KUKA KRL program: makrostep.src

&ACCESS RVP1
&COMMENT MAKRO_SCHRITTKETTE
&PARAM TEMPLATE = C:\KRC\Roboter\Template\makrostepvorgabe.src
&PARAM TPVW_VERSION = 8.1.8
&PARAM EDITMASK = MakroStep
DEF MAKROSTEP(Function :IN)
   ; FOLD Makro Schrittkette;%{SE} %MKUKATPVW
   ; FOLD ;%{H} %MKUKATPVW
   INT Function
   IF Function==1 THEN
     $APP_INT[5]=1
     Return
   ENDIF
   SWITCH $APP_INT[5]
   Case 0
   ; ENDFOLD
   ;ENDFOLD
   ;FOLD SCHRITT 1 -- -- ;%{P}%MKUKATPVW,%CSTEP,%VST_NR,%P 1:SCHRITT, 2:1, 3:
      ;FOLD ;%{H}
         Case 1
      ;ENDFOLD
      ;FOLD -- Roboter Schrittkette -- ;%{SE}%MKUKATPVW %CVW_COM %VCOMMENT %P 2:-- Roboter Schrittkette --, 3: VW_COMMENT
      ;ENDFOLD
      ;FOLD -- KS24 -- ;%{SE}%MKUKATPVW %CVW_COM %VCOMMENT %P 2:-- KS24 --, 3: VW_COMMENT
      ;ENDFOLD
      ;FOLD -- Version: 05 -- ;%{SE}%MKUKATPVW %CVW_COM %VCOMMENT %P 2:-- Version: 05 --, 3: VW_COMMENT
      ;ENDFOLD
      ;FOLD -- Stand: 001 -- ;%{SE}%MKUKATPVW %CVW_COM %VCOMMENT %P 2:-- Stand: 001 --, 3: VW_COMMENT
      ;ENDFOLD
      ;FOLD -- letzte Aenderung 24.10.2017 LZ -- ;%{SE}%MKUKATPVW %CVW_COM %VCOMMENT %P 2:-- letzte Aenderung 24.10.2017 LZ --, 3: VW_COMMENT
      ;ENDFOLD
      ;FOLD -- E/A's und Flags Ruecksetzen -- ;%{SE}%MKUKATPVW %CVW_COM %VCOMMENT %P 2:-- E/A's und Flags Ruecksetzen --, 3: VW_COMMENT
      ;ENDFOLD
      ;FOLD -- SK1 KF1 KS1 KE1 -- ;%{SE}%MKUKATPVW %CVW_COM %VCOMMENT %P 2:-- SK1 KF1 KS1 KE1 --, 3: VW_COMMENT
      ;ENDFOLD
      ;FOLD A786 = F830 & A786 ;%{SE}%MKUKATPVW %CVW_SPS %VBOASG %P 2:A786 = F830 & A786, 3: BOASG
         $OUT[786] = $FLAG[830] AND $OUT[786]
      ;ENDFOLD
      ;FOLD A722 = !F830 & A722 ;%{SE}%MKUKATPVW %CVW_SPS %VBOASG %P 2:A722 = !F830 & A722, 3: BOASG
         $OUT[722] = NOT $FLAG[830] AND $OUT[722]
      ;ENDFOLD
      ;FOLD A834 = AUS ;%{SE}%MKUKATPVW %CVW_SPS %VBOASG %P 2:A834 = AUS, 3: BOASG
         $OUT[834] = FALSE
      ;ENDFOLD
      ;FOLD A842 = AUS ;%{SE}%MKUKATPVW %CVW_SPS %VBOASG %P 2:A842 = AUS, 3: BOASG
         $OUT[842] = FALSE
      ;ENDFOLD
      ;FOLD -- SK2 KF2 KS2 KE2 -- ;%{SE}%MKUKATPVW %CVW_COM %VCOMMENT %P 2:-- SK2 KF2 KS2 KE2 --, 3: VW_COMMENT
      ;ENDFOLD
      ;FOLD A946 = F831 & A946 ;%{SE}%MKUKATPVW %CVW_SPS %VBOASG %P 2:A946 = F831 & A946, 3: BOASG
         $OUT[946] = $FLAG[831] AND $OUT[946]
      ;ENDFOLD
      ;FOLD A882 = !F831 & A882 ;%{SE}%MKUKATPVW %CVW_SPS %VBOASG %P 2:A882 = !F831 & A882, 3: BOASG
         $OUT[882] = NOT $FLAG[831] AND $OUT[882]
      ;ENDFOLD
      ;FOLD A994 = AUS ;%{SE}%MKUKATPVW %CVW_SPS %VBOASG %P 2:A994 = AUS, 3: BOASG
         $OUT[994] = FALSE
      ;ENDFOLD
      ;FOLD A995 = AUS ;%{SE}%MKUKATPVW %CVW_SPS %VBOASG %P 2:A995 = AUS, 3: BOASG
         $OUT[995] = FALSE
      ;ENDFOLD
      ;FOLD A1002 = AUS ;%{SE}%MKUKATPVW %CVW_SPS %VBOASG %P 2:A1002 = AUS, 3: BOASG
         $OUT[1002] = FALSE
      ;ENDFOLD
      ;FOLD -- SK3 KF3 KS3 KE3 -- ;%{SE}%MKUKATPVW %CVW_COM %VCOMMENT %P 2:-- SK3 KF3 KS3 KE3 --, 3: VW_COMMENT
      ;ENDFOLD
      ;FOLD A1106 = F832 & A1106 ;%{SE}%MKUKATPVW %CVW_SPS %VBOASG %P 2:A1106 = F832 & A1106, 3: BOASG
         $OUT[1106] = $FLAG[832] AND $OUT[1106]
      ;ENDFOLD
      ;FOLD A1042 = !F832 & A1042 ;%{SE}%MKUKATPVW %CVW_SPS %VBOASG %P 2:A1042 = !F832 & A1042, 3: BOASG
         $OUT[1042] = NOT $FLAG[832] AND $OUT[1042]
      ;ENDFOLD
      ;FOLD A1154 = AUS ;%{SE}%MKUKATPVW %CVW_SPS %VBOASG %P 2:A1154 = AUS, 3: BOASG
         $OUT[1154] = FALSE
      ;ENDFOLD
      ;FOLD A1155 = AUS ;%{SE}%MKUKATPVW %CVW_SPS %VBOASG %P 2:A1155 = AUS, 3: BOASG
         $OUT[1155] = FALSE
      ;ENDFOLD
      ;FOLD A1162 = AUS ;%{SE}%MKUKATPVW %CVW_SPS %VBOASG %P 2:A1162 = AUS, 3: BOASG
         $OUT[1162] = FALSE
      ;ENDFOLD
      ;FOLD -- Auswertung KF Umdrehungen EZ1/SP1/KE1 -- ;%{SE}%MKUKATPVW %CVW_COM %VCOMMENT %P 2:-- Auswertung KF Umdrehungen EZ1/SP1/KE1 --, 3: VW_COMMENT
      ;ENDFOLD
      ;FOLD F94 = AUS ;%{SE}%MKUKATPVW %CVW_SPS %VBOASG %P 2:F94 = AUS, 3: BOASG
         $FLAG[94] = FALSE
      ;ENDFOLD
      ;FOLD F95 = AUS ;%{SE}%MKUKATPVW %CVW_SPS %VBOASG %P 2:F95 = AUS, 3: BOASG
         $FLAG[95] = FALSE
      ;ENDFOLD
      ;FOLD F96 = AUS ;%{SE}%MKUKATPVW %CVW_SPS %VBOASG %P 2:F96 = AUS, 3: BOASG
         $FLAG[96] = FALSE
      ;ENDFOLD
      ;FOLD F97 = AUS ;%{SE}%MKUKATPVW %CVW_SPS %VBOASG %P 2:F97 = AUS, 3: BOASG
         $FLAG[97] = FALSE
      ;ENDFOLD
      ;FOLD F98 = AUS ;%{SE}%MKUKATPVW %CVW_SPS %VBOASG %P 2:F98 = AUS, 3: BOASG
         $FLAG[98] = FALSE
      ;ENDFOLD
      ;FOLD F99 = AUS ;%{SE}%MKUKATPVW %CVW_SPS %VBOASG %P 2:F99 = AUS, 3: BOASG
         $FLAG[99] = FALSE
      ;ENDFOLD
      ;FOLD F100 = AUS ;%{SE}%MKUKATPVW %CVW_SPS %VBOASG %P 2:F100 = AUS, 3: BOASG
         $FLAG[100] = FALSE
      ;ENDFOLD
      ;FOLD F101 = AUS ;%{SE}%MKUKATPVW %CVW_SPS %VBOASG %P 2:F101 = AUS, 3: BOASG
         $FLAG[101] = FALSE
      ;ENDFOLD
      ;FOLD F102 = AUS ;%{SE}%MKUKATPVW %CVW_SPS %VBOASG %P 2:F102 = AUS, 3: BOASG
         $FLAG[102] = FALSE
      ;ENDFOLD
      ;FOLD F103 = AUS ;%{SE}%MKUKATPVW %CVW_SPS %VBOASG %P 2:F103 = AUS, 3: BOASG
         $FLAG[103] = FALSE
      ;ENDFOLD
      ;FOLD F104 = AUS ;%{SE}%MKUKATPVW %CVW_SPS %VBOASG %P 2:F104 = AUS, 3: BOASG
         $FLAG[104] = FALSE
      ;ENDFOLD
      ;FOLD F105 = AUS ;%{SE}%MKUKATPVW %CVW_SPS %VBOASG %P 2:F105 = AUS, 3: BOASG
         $FLAG[105] = FALSE
      ;ENDFOLD
      ;FOLD F106 = AUS ;%{SE}%MKUKATPVW %CVW_SPS %VBOASG %P 2:F106 = AUS, 3: BOASG
         $FLAG[106] = FALSE
      ;ENDFOLD
      ;FOLD F107 = AUS ;%{SE}%MKUKATPVW %CVW_SPS %VBOASG %P 2:F107 = AUS, 3: BOASG
         $FLAG[107] = FALSE
      ;ENDFOLD
      ;FOLD F108 = AUS ;%{SE}%MKUKATPVW %CVW_SPS %VBOASG %P 2:F108 = AUS, 3: BOASG
         $FLAG[108] = FALSE
      ;ENDFOLD
      ;FOLD F109 = AUS ;%{SE}%MKUKATPVW %CVW_SPS %VBOASG %P 2:F109 = AUS, 3: BOASG
         $FLAG[109] = FALSE
      ;ENDFOLD
      ;FOLD F110 = AUS ;%{SE}%MKUKATPVW %CVW_SPS %VBOASG %P 2:F110 = AUS, 3: BOASG
         $FLAG[110] = FALSE
      ;ENDFOLD
      ;FOLD F111 = AUS ;%{SE}%MKUKATPVW %CVW_SPS %VBOASG %P 2:F111 = AUS, 3: BOASG
         $FLAG[111] = FALSE
      ;ENDFOLD
      ;FOLD F112 = AUS ;%{SE}%MKUKATPVW %CVW_SPS %VBOASG %P 2:F112 = AUS, 3: BOASG
         $FLAG[112] = FALSE
      ;ENDFOLD
      ;FOLD F113 = AUS ;%{SE}%MKUKATPVW %CVW_SPS %VBOASG %P 2:F113 = AUS, 3: BOASG
         $FLAG[113] = FALSE
      ;ENDFOLD
      ;FOLD F114 = AUS ;%{SE}%MKUKATPVW %CVW_SPS %VBOASG %P 2:F114 = AUS, 3: BOASG
         $FLAG[114] = FALSE
      ;ENDFOLD
      ;FOLD F115 = AUS ;%{SE}%MKUKATPVW %CVW_SPS %VBOASG %P 2:F115 = AUS, 3: BOASG
         $FLAG[115] = FALSE
      ;ENDFOLD
      ;FOLD F116 = AUS ;%{SE}%MKUKATPVW %CVW_SPS %VBOASG %P 2:F116 = AUS, 3: BOASG
         $FLAG[116] = FALSE
      ;ENDFOLD
      ;FOLD F117 = AUS ;%{SE}%MKUKATPVW %CVW_SPS %VBOASG %P 2:F117 = AUS, 3: BOASG
         $FLAG[117] = FALSE
      ;ENDFOLD
      ;FOLD -- Auswertung KF Umdrehungen EZ2/SP2/KE2 -- ;%{SE}%MKUKATPVW %CVW_COM %VCOMMENT %P 2:-- Auswertung KF Umdrehungen EZ2/SP2/KE2 --, 3: VW_COMMENT
      ;ENDFOLD
      ;FOLD F150 = AUS ;%{SE}%MKUKATPVW %CVW_SPS %VBOASG %P 2:F150 = AUS, 3: BOASG
         $FLAG[150] = FALSE
      ;ENDFOLD
      ;FOLD F151 = AUS ;%{SE}%MKUKATPVW %CVW_SPS %VBOASG %P 2:F151 = AUS, 3: BOASG
         $FLAG[151] = FALSE
      ;ENDFOLD
      ;FOLD F152 = AUS ;%{SE}%MKUKATPVW %CVW_SPS %VBOASG %P 2:F152 = AUS, 3: BOASG
         $FLAG[152] = FALSE
      ;ENDFOLD
      ;FOLD F153 = AUS ;%{SE}%MKUKATPVW %CVW_SPS %VBOASG %P 2:F153 = AUS, 3: BOASG
         $FLAG[153] = FALSE
      ;ENDFOLD
      ;FOLD F154 = AUS ;%{SE}%MKUKATPVW %CVW_SPS %VBOASG %P 2:F154 = AUS, 3: BOASG
         $FLAG[154] = FALSE
      ;ENDFOLD
      ;FOLD F155 = AUS ;%{SE}%MKUKATPVW %CVW_SPS %VBOASG %P 2:F155 = AUS, 3: BOASG
         $FLAG[155] = FALSE
      ;ENDFOLD
      ;FOLD -- Auswertung KF Umdrehungen EZ3/SP3/KE3 -- ;%{SE}%MKUKATPVW %CVW_COM %VCOMMENT %P 2:-- Auswertung KF Umdrehungen EZ3/SP3/KE3 --, 3: VW_COMMENT
      ;ENDFOLD
      ;FOLD F186 = AUS ;%{SE}%MKUKATPVW %CVW_SPS %VBOASG %P 2:F186 = AUS, 3: BOASG
         $FLAG[186] = FALSE
      ;ENDFOLD
      ;FOLD F187 = AUS ;%{SE}%MKUKATPVW %CVW_SPS %VBOASG %P 2:F187 = AUS, 3: BOASG
         $FLAG[187] = FALSE
      ;ENDFOLD
      ;FOLD F188 = AUS ;%{SE}%MKUKATPVW %CVW_SPS %VBOASG %P 2:F188 = AUS, 3: BOASG
         $FLAG[188] = FALSE
      ;ENDFOLD
      ;FOLD F189 = AUS ;%{SE}%MKUKATPVW %CVW_SPS %VBOASG %P 2:F189 = AUS, 3: BOASG
         $FLAG[189] = FALSE
      ;ENDFOLD
      ;FOLD F190 = AUS ;%{SE}%MKUKATPVW %CVW_SPS %VBOASG %P 2:F190 = AUS, 3: BOASG
         $FLAG[190] = FALSE
      ;ENDFOLD
      ;FOLD F191 = AUS ;%{SE}%MKUKATPVW %CVW_SPS %VBOASG %P 2:F191 = AUS, 3: BOASG
         $FLAG[191] = FALSE
      ;ENDFOLD
      ;FOLD -- Hilfsflags beim Fraesen -- ;%{SE}%MKUKATPVW %CVW_COM %VCOMMENT %P 2:-- Hilfsflags beim Fraesen --, 3: VW_COMMENT
      ;ENDFOLD
      ;FOLD F749 = AUS ;%{SE}%MKUKATPVW %CVW_SPS %VBOASG %P 2:F749 = AUS, 3: BOASG
         $FLAG[749] = FALSE
      ;ENDFOLD
      ;FOLD F287 = AUS ;%{SE}%MKUKATPVW %CVW_SPS %VBOASG %P 2:F287 = AUS, 3: BOASG
         $FLAG[287] = FALSE
      ;ENDFOLD
      ;FOLD F290 = AUS ;%{SE}%MKUKATPVW %CVW_SPS %VBOASG %P 2:F290 = AUS, 3: BOASG
         $FLAG[290] = FALSE
      ;ENDFOLD
      ;FOLD F291 = AUS ;%{SE}%MKUKATPVW %CVW_SPS %VBOASG %P 2:F291 = AUS, 3: BOASG
         $FLAG[291] = FALSE
      ;ENDFOLD
      ;FOLD -- Hilfsflags SZ2 an SK1 -- ;%{SE}%MKUKATPVW %CVW_COM %VCOMMENT %P 2:-- Hilfsflags SZ2 an SK1 --, 3: VW_COMMENT
      ;ENDFOLD
      ;FOLD F307 = AUS ;%{SE}%MKUKATPVW %CVW_SPS %VBOASG %P 2:F307 = AUS, 3: BOASG
         $FLAG[307] = FALSE
      ;ENDFOLD
      ;FOLD F308 = AUS ;%{SE}%MKUKATPVW %CVW_SPS %VBOASG %P 2:F308 = AUS, 3: BOASG
         $FLAG[308] = FALSE
      ;ENDFOLD
      ;FOLD -- Hilfsflags Funktionstest KF Motor -- ;%{SE}%MKUKATPVW %CVW_COM %VCOMMENT %P 2:-- Hilfsflags Funktionstest KF Motor --, 3: VW_COMMENT
      ;ENDFOLD
      ;FOLD F312 = AUS ;%{SE}%MKUKATPVW %CVW_SPS %VBOASG %P 2:F312 = AUS, 3: BOASG
         $FLAG[312] = FALSE
      ;ENDFOLD
      ;FOLD F313 = AUS ;%{SE}%MKUKATPVW %CVW_SPS %VBOASG %P 2:F313 = AUS, 3: BOASG
         $FLAG[313] = FALSE
      ;ENDFOLD
      ;FOLD -- RSK Fehlerausgaben -- ;%{SE}%MKUKATPVW %CVW_COM %VCOMMENT %P 2:-- RSK Fehlerausgaben --, 3: VW_COMMENT
      ;ENDFOLD
      ;FOLD F322 = AUS ;%{SE}%MKUKATPVW %CVW_SPS %VBOASG %P 2:F322 = AUS, 3: BOASG
         $FLAG[322] = FALSE
      ;ENDFOLD
      ;FOLD F323 = AUS ;%{SE}%MKUKATPVW %CVW_SPS %VBOASG %P 2:F323 = AUS, 3: BOASG
         $FLAG[323] = FALSE
      ;ENDFOLD
      ;FOLD F324 = AUS ;%{SE}%MKUKATPVW %CVW_SPS %VBOASG %P 2:F324 = AUS, 3: BOASG
         $FLAG[324] = FALSE
      ;ENDFOLD
      ;FOLD F325 = AUS ;%{SE}%MKUKATPVW %CVW_SPS %VBOASG %P 2:F325 = AUS, 3: BOASG
         $FLAG[325] = FALSE
      ;ENDFOLD
      ;FOLD F326 = AUS ;%{SE}%MKUKATPVW %CVW_SPS %VBOASG %P 2:F326 = AUS, 3: BOASG
         $FLAG[326] = FALSE
      ;ENDFOLD
      ;FOLD F327 = AUS ;%{SE}%MKUKATPVW %CVW_SPS %VBOASG %P 2:F327 = AUS, 3: BOASG
         $FLAG[327] = FALSE
      ;ENDFOLD
      ;FOLD F328 = AUS ;%{SE}%MKUKATPVW %CVW_SPS %VBOASG %P 2:F328 = AUS, 3: BOASG
         $FLAG[328] = FALSE
      ;ENDFOLD
      ;FOLD F329 = AUS ;%{SE}%MKUKATPVW %CVW_SPS %VBOASG %P 2:F329 = AUS, 3: BOASG
         $FLAG[329] = FALSE
      ;ENDFOLD
      ;FOLD -- Hilfsflag SK Programmwechsel -- ;%{SE}%MKUKATPVW %CVW_COM %VCOMMENT %P 2:-- Hilfsflag SK Programmwechsel --, 3: VW_COMMENT
      ;ENDFOLD
      ;FOLD F334 = AUS ;%{SE}%MKUKATPVW %CVW_SPS %VBOASG %P 2:F334 = AUS, 3: BOASG
         $FLAG[334] = FALSE
      ;ENDFOLD
      ;FOLD -- Flag KL1 Spueleimer -- ;%{SE}%MKUKATPVW %CVW_COM %VCOMMENT %P 2:-- Flag KL1 Spueleimer --, 3: VW_COMMENT
      ;ENDFOLD
      ;FOLD F352 = AUS ;%{SE}%MKUKATPVW %CVW_SPS %VBOASG %P 2:F352 = AUS, 3: BOASG
         $FLAG[352] = FALSE
      ;ENDFOLD
      ;FOLD F353 = AUS ;%{SE}%MKUKATPVW %CVW_SPS %VBOASG %P 2:F353 = AUS, 3: BOASG
         $FLAG[353] = FALSE
      ;ENDFOLD
      ;FOLD -- Flag KL2 Spueleimer -- ;%{SE}%MKUKATPVW %CVW_COM %VCOMMENT %P 2:-- Flag KL2 Spueleimer --, 3: VW_COMMENT
      ;ENDFOLD
      ;FOLD F373 = AUS ;%{SE}%MKUKATPVW %CVW_SPS %VBOASG %P 2:F373 = AUS, 3: BOASG
         $FLAG[373] = FALSE
      ;ENDFOLD
      ;FOLD F374 = AUS ;%{SE}%MKUKATPVW %CVW_SPS %VBOASG %P 2:F374 = AUS, 3: BOASG
         $FLAG[374] = FALSE
      ;ENDFOLD
      ;FOLD -- Flag KL3 Spueleimer -- ;%{SE}%MKUKATPVW %CVW_COM %VCOMMENT %P 2:-- Flag KL3 Spueleimer --, 3: VW_COMMENT
      ;ENDFOLD
      ;FOLD F394 = AUS ;%{SE}%MKUKATPVW %CVW_SPS %VBOASG %P 2:F394 = AUS, 3: BOASG
         $FLAG[394] = FALSE
      ;ENDFOLD
      ;FOLD F395 = AUS ;%{SE}%MKUKATPVW %CVW_SPS %VBOASG %P 2:F395 = AUS, 3: BOASG
         $FLAG[395] = FALSE
      ;ENDFOLD
      ;FOLD -- Flag MS Reinigung gestartet -- ;%{SE}%MKUKATPVW %CVW_COM %VCOMMENT %P 2:-- Flag MS Reinigung gestartet --, 3: VW_COMMENT
      ;ENDFOLD
      ;FOLD F604 = AUS ;%{SE}%MKUKATPVW %CVW_SPS %VBOASG %P 2:F604 = AUS, 3: BOASG
         $FLAG[604] = FALSE
      ;ENDFOLD
      ;FOLD F608 = AUS ;%{SE}%MKUKATPVW %CVW_SPS %VBOASG %P 2:F608 = AUS, 3: BOASG
         $FLAG[608] = FALSE
      ;ENDFOLD
      ;FOLD -- Timer Stoppen -- ;%{SE}%MKUKATPVW %CVW_COM %VCOMMENT %P 2:-- Timer Stoppen --, 3: VW_COMMENT
      ;ENDFOLD
      ;FOLD t7 ( EIN ) = STOP ;%{SE}%MKUKATPVW %CVW_SPS %VTSTOP %P 2:t7 ( EIN ) = STOP, 3: TSTOP
         VW(#SET_TIME,TRUE,7,1,0)
      ;ENDFOLD
      ;FOLD t8 ( EIN ) = STOP ;%{SE}%MKUKATPVW %CVW_SPS %VTSTOP %P 2:t8 ( EIN ) = STOP, 3: TSTOP
         VW(#SET_TIME,TRUE,8,1,0)
      ;ENDFOLD
      ;FOLD t9 ( EIN ) = STOP ;%{SE}%MKUKATPVW %CVW_SPS %VTSTOP %P 2:t9 ( EIN ) = STOP, 3: TSTOP
         VW(#SET_TIME,TRUE,9,1,0)
      ;ENDFOLD
      ;FOLD Schritt 2 = EIN  ;%{SE}%MKUKATPVW %CVW_SPS %VST_CON %P 2:Schritt 2 = EIN , 3: ST_CON
         IF TRUE THEN
            PREVSTEP = $APP_INT[5]
            $APP_INT[5] = 2
         ENDIF
      ;ENDFOLD
   ;ENDFOLD
   ;FOLD SCHRITT 2 -- RSK Grundstellung # Anwahlen-- ;%{P}%MKUKATPVW,%CSTEP,%VST_NR,%P 1:SCHRITT, 2:2, 3: RSK Grundstellung # Anwahlen
      ;FOLD ;%{H}
         Case 2
      ;ENDFOLD
      ;FOLD -- RSK in Grundstellung -- ;%{SE}%MKUKATPVW %CVW_COM %VCOMMENT %P 2:-- RSK in Grundstellung --, 3: VW_COMMENT
      ;ENDFOLD
      ;FOLD F321 = EIN ;%{SE}%MKUKATPVW %CVW_SPS %VBOASG %P 2:F321 = EIN, 3: BOASG
         $FLAG[321] = TRUE
      ;ENDFOLD
      ;FOLD -- Fraesen ROB EZ1/SP1/KE1 SZ1 (Basic/Docking) -- ;%{SE}%MKUKATPVW %CVW_COM %VCOMMENT %P 2:-- Fraesen ROB EZ1/SP1/KE1 SZ1 (Basic/Docking) --, 3: VW_COMMENT
      ;ENDFOLD
      ;FOLD Schritt 3 = F64 & !F65 & !F66 & !F67 & F90 & !F91 & !F565 & A4039  ;%{SE}%MKUKATPVW %CVW_SPS %VST_CON %P 2:Schritt 3 = F64 & !F65 & !F66 & !F67 & F90 & !F91 & !F565 & A4039 , 3: ST_CON
         IF $FLAG[64] AND NOT $FLAG[65] AND NOT $FLAG[66] AND NOT $FLAG[67] AND $FLAG[90] AND NOT $FLAG[91] AND NOT $FLAG[565] AND $OUT[4039] THEN
            PREVSTEP = $APP_INT[5]
            $APP_INT[5] = 3
         ENDIF
      ;ENDFOLD
      ;FOLD -- Fraesen ROB EZ1/SP1/KE1 SZ2 (Docking) -- ;%{SE}%MKUKATPVW %CVW_COM %VCOMMENT %P 2:-- Fraesen ROB EZ1/SP1/KE1 SZ2 (Docking) --, 3: VW_COMMENT
      ;ENDFOLD
      ;FOLD Schritt 15 = !F64 & F65 & !F66 & !F67 & F90 & !F91 & !F565 & A4039  ;%{SE}%MKUKATPVW %CVW_SPS %VST_CON %P 2:Schritt 15 = !F64 & F65 & !F66 & !F67 & F90 & !F91 & !F565 & A4039 , 3: ST_CON
         IF NOT $FLAG[64] AND $FLAG[65] AND NOT $FLAG[66] AND NOT $FLAG[67] AND $FLAG[90] AND NOT $FLAG[91] AND NOT $FLAG[565] AND $OUT[4039] THEN
            PREVSTEP = $APP_INT[5]
            $APP_INT[5] = 15
         ENDIF
      ;ENDFOLD
      ;FOLD -- Fraesen ROB EZ1/SP1/KE1 SZ3 (Docking) -- ;%{SE}%MKUKATPVW %CVW_COM %VCOMMENT %P 2:-- Fraesen ROB EZ1/SP1/KE1 SZ3 (Docking) --, 3: VW_COMMENT
      ;ENDFOLD
      ;FOLD Schritt 27 = !F64 & !F65 & F66 & !F67 & F90 & !F91 & !F565 & A4039  ;%{SE}%MKUKATPVW %CVW_SPS %VST_CON %P 2:Schritt 27 = !F64 & !F65 & F66 & !F67 & F90 & !F91 & !F565 & A4039 , 3: ST_CON
         IF NOT $FLAG[64] AND NOT $FLAG[65] AND $FLAG[66] AND NOT $FLAG[67] AND $FLAG[90] AND NOT $FLAG[91] AND NOT $FLAG[565] AND $OUT[4039] THEN
            PREVSTEP = $APP_INT[5]
            $APP_INT[5] = 27
         ENDIF
      ;ENDFOLD
      ;FOLD -- Fraesen ROB EZ1/SP1/KE1 SZ4 (Docking) -- ;%{SE}%MKUKATPVW %CVW_COM %VCOMMENT %P 2:-- Fraesen ROB EZ1/SP1/KE1 SZ4 (Docking) --, 3: VW_COMMENT
      ;ENDFOLD
      ;FOLD Schritt 39 = !F64 & !F65 & !F66 & F67 & F90 & !F91 & !F565 & A4039  ;%{SE}%MKUKATPVW %CVW_SPS %VST_CON %P 2:Schritt 39 = !F64 & !F65 & !F66 & F67 & F90 & !F91 & !F565 & A4039 , 3: ST_CON
         IF NOT $FLAG[64] AND NOT $FLAG[65] AND NOT $FLAG[66] AND $FLAG[67] AND $FLAG[90] AND NOT $FLAG[91] AND NOT $FLAG[565] AND $OUT[4039] THEN
            PREVSTEP = $APP_INT[5]
            $APP_INT[5] = 39
         ENDIF
      ;ENDFOLD
      ;FOLD -- Fraesen STAT EZ1/SP1/KE1 -- ;%{SE}%MKUKATPVW %CVW_COM %VCOMMENT %P 2:-- Fraesen STAT EZ1/SP1/KE1 --, 3: VW_COMMENT
      ;ENDFOLD
      ;FOLD Schritt 51 = F92 & !F93 & A4039 & E13  ;%{SE}%MKUKATPVW %CVW_SPS %VST_CON %P 2:Schritt 51 = F92 & !F93 & A4039 & E13 , 3: ST_CON
         IF $FLAG[92] AND NOT $FLAG[93] AND $OUT[4039] AND $IN[13] THEN
            PREVSTEP = $APP_INT[5]
            $APP_INT[5] = 51
         ENDIF
      ;ENDFOLD
      ;FOLD -- Fraesen STAT EZ2/SP2/KE2 -- ;%{SE}%MKUKATPVW %CVW_COM %VCOMMENT %P 2:-- Fraesen STAT EZ2/SP2/KE2 --, 3: VW_COMMENT
      ;ENDFOLD
      ;FOLD Schritt 74 = F148 & !F149 & A4039 & E13  ;%{SE}%MKUKATPVW %CVW_SPS %VST_CON %P 2:Schritt 74 = F148 & !F149 & A4039 & E13 , 3: ST_CON
         IF $FLAG[148] AND NOT $FLAG[149] AND $OUT[4039] AND $IN[13] THEN
            PREVSTEP = $APP_INT[5]
            $APP_INT[5] = 74
         ENDIF
      ;ENDFOLD
      ;FOLD -- Fraesen STAT EZ3/SP3/KE3 -- ;%{SE}%MKUKATPVW %CVW_COM %VCOMMENT %P 2:-- Fraesen STAT EZ3/SP3/KE3 --, 3: VW_COMMENT
      ;ENDFOLD
      ;FOLD Schritt 97 = F184 & !F185 & A4039 & E13  ;%{SE}%MKUKATPVW %CVW_SPS %VST_CON %P 2:Schritt 97 = F184 & !F185 & A4039 & E13 , 3: ST_CON
         IF $FLAG[184] AND NOT $FLAG[185] AND $OUT[4039] AND $IN[13] THEN
            PREVSTEP = $APP_INT[5]
            $APP_INT[5] = 97
         ENDIF
      ;ENDFOLD
      ;FOLD -- Fraesen ROB STP1 SZ1 (Stosspunkten) -- ;%{SE}%MKUKATPVW %CVW_COM %VCOMMENT %P 2:-- Fraesen ROB STP1 SZ1 (Stosspunkten) --, 3: VW_COMMENT
      ;ENDFOLD
      ;FOLD Schritt 120 = F64 & !F65 & !F66 & !F67 & F90 & !F91 & !F805 & F565 & A4039 & E13  ;%{SE}%MKUKATPVW %CVW_SPS %VST_CON %P 2:Schritt 120 = F64 & !F65 & !F66 & !F67 & F90 & !F91 & !F805 & F565 & A4039 & E13 , 3: ST_CON
         IF $FLAG[64] AND NOT $FLAG[65] AND NOT $FLAG[66] AND NOT $FLAG[67] AND $FLAG[90] AND NOT $FLAG[91] AND NOT $FLAG[805] AND $FLAG[565] AND $OUT[4039] AND $IN[13] THEN
            PREVSTEP = $APP_INT[5]
            $APP_INT[5] = 120
         ENDIF
      ;ENDFOLD
      ;FOLD -- MS1 Reinigung (an KS3 Schwenkeinheit) -- ;%{SE}%MKUKATPVW %CVW_COM %VCOMMENT %P 2:-- MS1 Reinigung (an KS3 Schwenkeinheit) --, 3: VW_COMMENT
      ;ENDFOLD
      ;FOLD Schritt 128 = F603 & !F605 & F528 & !F529 & A4039 & E13  ;%{SE}%MKUKATPVW %CVW_SPS %VST_CON %P 2:Schritt 128 = F603 & !F605 & F528 & !F529 & A4039 & E13 , 3: ST_CON
         IF $FLAG[603] AND NOT $FLAG[605] AND $FLAG[528] AND NOT $FLAG[529] AND $OUT[4039] AND $IN[13] THEN
            PREVSTEP = $APP_INT[5]
            $APP_INT[5] = 128
         ENDIF
      ;ENDFOLD
      ;FOLD -- MS2 Reinigung (an KS2 Schwenkeinheit) -- ;%{SE}%MKUKATPVW %CVW_COM %VCOMMENT %P 2:-- MS2 Reinigung (an KS2 Schwenkeinheit) --, 3: VW_COMMENT
      ;ENDFOLD
      ;FOLD Schritt 141 = F607 & !F609 & F528 & !F529 & A4039 & E13  ;%{SE}%MKUKATPVW %CVW_SPS %VST_CON %P 2:Schritt 141 = F607 & !F609 & F528 & !F529 & A4039 & E13 , 3: ST_CON
         IF $FLAG[607] AND NOT $FLAG[609] AND $FLAG[528] AND NOT $FLAG[529] AND $OUT[4039] AND $IN[13] THEN
            PREVSTEP = $APP_INT[5]
            $APP_INT[5] = 141
         ENDIF
      ;ENDFOLD
      ;FOLD -- MS1 Reinigung (an Pneum. Schwenkeinheit MS1) -- ;%{SE}%MKUKATPVW %CVW_COM %VCOMMENT %P 2:-- MS1 Reinigung (an Pneum. Schwenkeinheit MS1) --, 3: VW_COMMENT
      ;ENDFOLD
      ;FOLD Schritt 154 = F603 & !F605 & !F528 & F529 & A4039 & E13  ;%{SE}%MKUKATPVW %CVW_SPS %VST_CON %P 2:Schritt 154 = F603 & !F605 & !F528 & F529 & A4039 & E13 , 3: ST_CON
         IF $FLAG[603] AND NOT $FLAG[605] AND NOT $FLAG[528] AND $FLAG[529] AND $OUT[4039] AND $IN[13] THEN
            PREVSTEP = $APP_INT[5]
            $APP_INT[5] = 154
         ENDIF
      ;ENDFOLD
      ;FOLD -- MS2 Reinigung (an Pneum. Schwenkeinheit MS2) -- ;%{SE}%MKUKATPVW %CVW_COM %VCOMMENT %P 2:-- MS2 Reinigung (an Pneum. Schwenkeinheit MS2) --, 3: VW_COMMENT
      ;ENDFOLD
      ;FOLD Schritt 169 = F607 & !F609 & !F528 & F529 & A4039 & E13  ;%{SE}%MKUKATPVW %CVW_SPS %VST_CON %P 2:Schritt 169 = F607 & !F609 & !F528 & F529 & A4039 & E13 , 3: ST_CON
         IF $FLAG[607] AND NOT $FLAG[609] AND NOT $FLAG[528] AND $FLAG[529] AND $OUT[4039] AND $IN[13] THEN
            PREVSTEP = $APP_INT[5]
            $APP_INT[5] = 169
         ENDIF
      ;ENDFOLD
      ;FOLD -- KL1 Spueleimer (an Pneum. Schwenkeinheit KL1) -- ;%{SE}%MKUKATPVW %CVW_COM %VCOMMENT %P 2:-- KL1 Spueleimer (an Pneum. Schwenkeinheit KL1) --, 3: VW_COMMENT
      ;ENDFOLD
      ;FOLD -- in Arbeitsstellung schwenken -- ;%{SE}%MKUKATPVW %CVW_COM %VCOMMENT %P 2:-- in Arbeitsstellung schwenken --, 3: VW_COMMENT
      ;ENDFOLD
      ;FOLD Schritt 184 = !F352 & F353 & !F355 & (F523 & !F524 + !F523 & F524) & A4039 & E13  ;%{SE}%MKUKATPVW %CVW_SPS %VST_CON %P 2:Schritt 184 = !F352 & F353 & !F355 & (F523 & !F524 + !F523 & F524) & A4039 & E13 , 3: ST_CON
         IF NOT $FLAG[352] AND $FLAG[353] AND NOT $FLAG[355] AND ($FLAG[523] AND NOT $FLAG[524] OR NOT $FLAG[523] AND $FLAG[524]) AND $OUT[4039] AND $IN[13] THEN
            PREVSTEP = $APP_INT[5]
            $APP_INT[5] = 184
         ENDIF
      ;ENDFOLD
      ;FOLD -- KL1 Spueleimer (an Pneum. Schwenkeinheit KL1) -- ;%{SE}%MKUKATPVW %CVW_COM %VCOMMENT %P 2:-- KL1 Spueleimer (an Pneum. Schwenkeinheit KL1) --, 3: VW_COMMENT
      ;ENDFOLD
      ;FOLD -- in Ruhestellung schwenken -- ;%{SE}%MKUKATPVW %CVW_COM %VCOMMENT %P 2:-- in Ruhestellung schwenken --, 3: VW_COMMENT
      ;ENDFOLD
      ;FOLD Schritt 189 = F352 & !F353 & !F355 & (F523 & !F524 + !F523 & F524) & A4039 & E13  ;%{SE}%MKUKATPVW %CVW_SPS %VST_CON %P 2:Schritt 189 = F352 & !F353 & !F355 & (F523 & !F524 + !F523 & F524) & A4039 & E13 , 3: ST_CON
         IF $FLAG[352] AND NOT $FLAG[353] AND NOT $FLAG[355] AND ($FLAG[523] AND NOT $FLAG[524] OR NOT $FLAG[523] AND $FLAG[524]) AND $OUT[4039] AND $IN[13] THEN
            PREVSTEP = $APP_INT[5]
            $APP_INT[5] = 189
         ENDIF
      ;ENDFOLD
      ;FOLD -- KL2 Spueleimer (an Pneum. Schwenkeinheit KL2) -- ;%{SE}%MKUKATPVW %CVW_COM %VCOMMENT %P 2:-- KL2 Spueleimer (an Pneum. Schwenkeinheit KL2) --, 3: VW_COMMENT
      ;ENDFOLD
      ;FOLD -- in Arbeitsstellung schwenken -- ;%{SE}%MKUKATPVW %CVW_COM %VCOMMENT %P 2:-- in Arbeitsstellung schwenken --, 3: VW_COMMENT
      ;ENDFOLD
      ;FOLD Schritt 195 = !F373 & F374 & !F376 & (F523 & !F524 + !F523 & F524) & A4039 & E13  ;%{SE}%MKUKATPVW %CVW_SPS %VST_CON %P 2:Schritt 195 = !F373 & F374 & !F376 & (F523 & !F524 + !F523 & F524) & A4039 & E13 , 3: ST_CON
         IF NOT $FLAG[373] AND $FLAG[374] AND NOT $FLAG[376] AND ($FLAG[523] AND NOT $FLAG[524] OR NOT $FLAG[523] AND $FLAG[524]) AND $OUT[4039] AND $IN[13] THEN
            PREVSTEP = $APP_INT[5]
            $APP_INT[5] = 195
         ENDIF
      ;ENDFOLD
      ;FOLD -- KL2 Spueleimer (an Pneum. Schwenkeinheit KL2) -- ;%{SE}%MKUKATPVW %CVW_COM %VCOMMENT %P 2:-- KL2 Spueleimer (an Pneum. Schwenkeinheit KL2) --, 3: VW_COMMENT
      ;ENDFOLD
      ;FOLD -- in Ruhestellung schwenken -- ;%{SE}%MKUKATPVW %CVW_COM %VCOMMENT %P 2:-- in Ruhestellung schwenken --, 3: VW_COMMENT
      ;ENDFOLD
      ;FOLD Schritt 200 = F373 & !F374 & !F376 & (F523 & !F524 + !F523 & F524) & A4039 & E13  ;%{SE}%MKUKATPVW %CVW_SPS %VST_CON %P 2:Schritt 200 = F373 & !F374 & !F376 & (F523 & !F524 + !F523 & F524) & A4039 & E13 , 3: ST_CON
         IF $FLAG[373] AND NOT $FLAG[374] AND NOT $FLAG[376] AND ($FLAG[523] AND NOT $FLAG[524] OR NOT $FLAG[523] AND $FLAG[524]) AND $OUT[4039] AND $IN[13] THEN
            PREVSTEP = $APP_INT[5]
            $APP_INT[5] = 200
         ENDIF
      ;ENDFOLD
      ;FOLD -- KL3 Spueleimer (an Pneum. Schwenkeinheit KL3) -- ;%{SE}%MKUKATPVW %CVW_COM %VCOMMENT %P 2:-- KL3 Spueleimer (an Pneum. Schwenkeinheit KL3) --, 3: VW_COMMENT
      ;ENDFOLD
      ;FOLD -- in Arbeitsstellung schwenken -- ;%{SE}%MKUKATPVW %CVW_COM %VCOMMENT %P 2:-- in Arbeitsstellung schwenken --, 3: VW_COMMENT
      ;ENDFOLD
      ;FOLD Schritt 206 = !F394 & F395 & !F397 & (F523 & !F524 + !F523 & F524) & A4039 & E13  ;%{SE}%MKUKATPVW %CVW_SPS %VST_CON %P 2:Schritt 206 = !F394 & F395 & !F397 & (F523 & !F524 + !F523 & F524) & A4039 & E13 , 3: ST_CON
         IF NOT $FLAG[394] AND $FLAG[395] AND NOT $FLAG[397] AND ($FLAG[523] AND NOT $FLAG[524] OR NOT $FLAG[523] AND $FLAG[524]) AND $OUT[4039] AND $IN[13] THEN
            PREVSTEP = $APP_INT[5]
            $APP_INT[5] = 206
         ENDIF
      ;ENDFOLD
      ;FOLD -- KL3 Spueleimer (an Pneum. Schwenkeinheit KL3) -- ;%{SE}%MKUKATPVW %CVW_COM %VCOMMENT %P 2:-- KL3 Spueleimer (an Pneum. Schwenkeinheit KL3) --, 3: VW_COMMENT
      ;ENDFOLD
      ;FOLD -- in Ruhestellung schwenken -- ;%{SE}%MKUKATPVW %CVW_COM %VCOMMENT %P 2:-- in Ruhestellung schwenken --, 3: VW_COMMENT
      ;ENDFOLD
      ;FOLD Schritt 211 = F394 & !F395 & !F397 & (F523 & !F524 + !F523 & F524) & A4039 & E13  ;%{SE}%MKUKATPVW %CVW_SPS %VST_CON %P 2:Schritt 211 = F394 & !F395 & !F397 & (F523 & !F524 + !F523 & F524) & A4039 & E13 , 3: ST_CON
         IF $FLAG[394] AND NOT $FLAG[395] AND NOT $FLAG[397] AND ($FLAG[523] AND NOT $FLAG[524] OR NOT $FLAG[523] AND $FLAG[524]) AND $OUT[4039] AND $IN[13] THEN
            PREVSTEP = $APP_INT[5]
            $APP_INT[5] = 211
         ENDIF
      ;ENDFOLD
      ;FOLD -- Fraesen MB1 (an KSB1 Schwenkeinheit) -- ;%{SE}%MKUKATPVW %CVW_COM %VCOMMENT %P 2:-- Fraesen MB1 (an KSB1 Schwenkeinheit) --, 3: VW_COMMENT
      ;ENDFOLD
      ;FOLD Schritt 250 = F209 & !F210 & A4039 & E13  ;%{SE}%MKUKATPVW %CVW_SPS %VST_CON %P 2:Schritt 250 = F209 & !F210 & A4039 & E13 , 3: ST_CON
         IF $FLAG[209] AND NOT $FLAG[210] AND $OUT[4039] AND $IN[13] THEN
            PREVSTEP = $APP_INT[5]
            $APP_INT[5] = 250
         ENDIF
      ;ENDFOLD
      ;FOLD -- Fraesen ROB STP1 SZ1 (Stosspunkten & KW Braeuer) -- ;%{SE}%MKUKATPVW %CVW_COM %VCOMMENT %P 2:-- Fraesen ROB STP1 SZ1 (Stosspunkten & KW Braeuer) --, 3: VW_COMMENT
      ;ENDFOLD
      ;FOLD Schritt 272 = F64 & !F65 & !F66 & !F67 & F90 & !F91 & F805 & F565 & A4039  ;%{SE}%MKUKATPVW %CVW_SPS %VST_CON %P 2:Schritt 272 = F64 & !F65 & !F66 & !F67 & F90 & !F91 & F805 & F565 & A4039 , 3: ST_CON
         IF $FLAG[64] AND NOT $FLAG[65] AND NOT $FLAG[66] AND NOT $FLAG[67] AND $FLAG[90] AND NOT $FLAG[91] AND $FLAG[805] AND $FLAG[565] AND $OUT[4039] THEN
            PREVSTEP = $APP_INT[5]
            $APP_INT[5] = 272
         ENDIF
      ;ENDFOLD
   ;ENDFOLD
   ;FOLD SCHRITT 3 -- ROB EZ1/SP1/KE1 SZ1 # Start -- ;%{P}%MKUKATPVW,%CSTEP,%VST_NR,%P 1:SCHRITT, 2:3, 3: ROB EZ1/SP1/KE1 SZ1 # Start
      ;FOLD ;%{H}
         Case 3
      ;ENDFOLD
      ;FOLD -- RSK gestartet -- ;%{SE}%MKUKATPVW %CVW_COM %VCOMMENT %P 2:-- RSK gestartet --, 3: VW_COMMENT
      ;ENDFOLD
      ;FOLD F321 = AUS ;%{SE}%MKUKATPVW %CVW_SPS %VBOASG %P 2:F321 = AUS, 3: BOASG
         $FLAG[321] = FALSE
      ;ENDFOLD
      ;FOLD F322 = AUS ;%{SE}%MKUKATPVW %CVW_SPS %VBOASG %P 2:F322 = AUS, 3: BOASG
         $FLAG[322] = FALSE
      ;ENDFOLD
      ;FOLD F323 = AUS ;%{SE}%MKUKATPVW %CVW_SPS %VBOASG %P 2:F323 = AUS, 3: BOASG
         $FLAG[323] = FALSE
      ;ENDFOLD
      ;FOLD F324 = AUS ;%{SE}%MKUKATPVW %CVW_SPS %VBOASG %P 2:F324 = AUS, 3: BOASG
         $FLAG[324] = FALSE
      ;ENDFOLD
      ;FOLD F325 = AUS ;%{SE}%MKUKATPVW %CVW_SPS %VBOASG %P 2:F325 = AUS, 3: BOASG
         $FLAG[325] = FALSE
      ;ENDFOLD
      ;FOLD F327 = AUS ;%{SE}%MKUKATPVW %CVW_SPS %VBOASG %P 2:F327 = AUS, 3: BOASG
         $FLAG[327] = FALSE
      ;ENDFOLD
      ;FOLD F329 = AUS ;%{SE}%MKUKATPVW %CVW_SPS %VBOASG %P 2:F329 = AUS, 3: BOASG
         $FLAG[329] = FALSE
      ;ENDFOLD
      ;FOLD -- EZ1/SP1/KE1 SZ1 Zaehler -- ;%{SE}%MKUKATPVW %CVW_COM %VCOMMENT %P 2:-- EZ1/SP1/KE1 SZ1 Zaehler --, 3: VW_COMMENT
      ;ENDFOLD
      ;FOLD F94 = AUS ;%{SE}%MKUKATPVW %CVW_SPS %VBOASG %P 2:F94 = AUS, 3: BOASG
         $FLAG[94] = FALSE
      ;ENDFOLD
      ;FOLD F95 = AUS ;%{SE}%MKUKATPVW %CVW_SPS %VBOASG %P 2:F95 = AUS, 3: BOASG
         $FLAG[95] = FALSE
      ;ENDFOLD
      ;FOLD F96 = AUS ;%{SE}%MKUKATPVW %CVW_SPS %VBOASG %P 2:F96 = AUS, 3: BOASG
         $FLAG[96] = FALSE
      ;ENDFOLD
      ;FOLD F97 = AUS ;%{SE}%MKUKATPVW %CVW_SPS %VBOASG %P 2:F97 = AUS, 3: BOASG
         $FLAG[97] = FALSE
      ;ENDFOLD
      ;FOLD F98 = AUS ;%{SE}%MKUKATPVW %CVW_SPS %VBOASG %P 2:F98 = AUS, 3: BOASG
         $FLAG[98] = FALSE
      ;ENDFOLD
      ;FOLD F99 = AUS ;%{SE}%MKUKATPVW %CVW_SPS %VBOASG %P 2:F99 = AUS, 3: BOASG
         $FLAG[99] = FALSE
      ;ENDFOLD
      ;FOLD -- Hilfsflags KF/KW1 Motor/Initiator -- ;%{SE}%MKUKATPVW %CVW_COM %VCOMMENT %P 2:-- Hilfsflags KF/KW1 Motor/Initiator --, 3: VW_COMMENT
      ;ENDFOLD
      ;FOLD F312 = AUS ;%{SE}%MKUKATPVW %CVW_SPS %VBOASG %P 2:F312 = AUS, 3: BOASG
         $FLAG[312] = FALSE
      ;ENDFOLD
      ;FOLD F313 = AUS ;%{SE}%MKUKATPVW %CVW_SPS %VBOASG %P 2:F313 = AUS, 3: BOASG
         $FLAG[313] = FALSE
      ;ENDFOLD
      ;FOLD -- Rob. EZ1/SP1/KE1 SZ1 beim Fraesen -- ;%{SE}%MKUKATPVW %CVW_COM %VCOMMENT %P 2:-- Rob. EZ1/SP1/KE1 SZ1 beim Fraesen --, 3: VW_COMMENT
      ;ENDFOLD
      ;FOLD A116 = EIN ;%{SE}%MKUKATPVW %CVW_SPS %VBOASG %P 2:A116 = EIN, 3: BOASG
         $OUT[116] = TRUE
      ;ENDFOLD
      ;FOLD A130 = EIN ;%{SE}%MKUKATPVW %CVW_SPS %VBOASG %P 2:A130 = EIN, 3: BOASG
         $OUT[130] = TRUE
      ;ENDFOLD
      ;FOLD -- Quitt. Fraesen SK1 AUS -- ;%{SE}%MKUKATPVW %CVW_COM %VCOMMENT %P 2:-- Quitt. Fraesen SK1 AUS --, 3: VW_COMMENT
      ;ENDFOLD
      ;FOLD A786 = F830 & A786 ;%{SE}%MKUKATPVW %CVW_SPS %VBOASG %P 2:A786 = F830 & A786, 3: BOASG
         $OUT[786] = $FLAG[830] AND $OUT[786]
      ;ENDFOLD
      ;FOLD -- Ueberwachungszeit KF1/KW1 -- ;%{SE}%MKUKATPVW %CVW_COM %VCOMMENT %P 2:-- Ueberwachungszeit KF1/KW1 --, 3: VW_COMMENT
      ;ENDFOLD
      ;FOLD t7 ( EIN ) = -30[1/10Sek] ;%{SE}%MKUKATPVW %CVW_SPS %VTASG %P 2:t7 ( EIN ) = -30[1/10Sek], 3: TASG
         VW(#SET_TIME,TRUE,7,0,-30)
      ;ENDFOLD
      ;FOLD Schritt 4 = A4039  ;%{SE}%MKUKATPVW %CVW_SPS %VST_CON %P 2:Schritt 4 = A4039 , 3: ST_CON
         IF $OUT[4039] THEN
            PREVSTEP = $APP_INT[5]
            $APP_INT[5] = 4
         ENDIF
      ;ENDFOLD
   ;ENDFOLD
   ;FOLD SCHRITT 4 -- ROB EZ1/SP1/KE1 SZ1 -- ;%{P}%MKUKATPVW,%CSTEP,%VST_NR,%P 1:SCHRITT, 2:4, 3: ROB EZ1/SP1/KE1 SZ1
      ;FOLD ;%{H}
         Case 4
      ;ENDFOLD
      ;FOLD -- KF1/KW1 einschalten -- ;%{SE}%MKUKATPVW %CVW_COM %VCOMMENT %P 2:-- KF1/KW1 einschalten --, 3: VW_COMMENT
      ;ENDFOLD
      ;FOLD i1 (EIN) = 0 ;%{SE}%MKUKATPVW %CVW_SPS %VARIASG %P 2:i1 (EIN) = 0, 3: ARIASG
         VW(#COUNTER,TRUE,1,0)
      ;ENDFOLD
      ;FOLD A834 = !F289 ;%{SE}%MKUKATPVW %CVW_SPS %VBOASG %P 2:A834 = !F289, 3: BOASG
         $OUT[834] = NOT $FLAG[289]
      ;ENDFOLD
      ;FOLD A858 = F289 ;%{SE}%MKUKATPVW %CVW_SPS %VBOASG %P 2:A858 = F289, 3: BOASG
         $OUT[858] = $FLAG[289]
      ;ENDFOLD
      ;FOLD A1018 = F803 ;%{SE}%MKUKATPVW %CVW_SPS %VBOASG %P 2:A1018 = F803, 3: BOASG
         $OUT[1018] = $FLAG[803]
      ;ENDFOLD
      ;FOLD Schritt 5 = A4039  ;%{SE}%MKUKATPVW %CVW_SPS %VST_CON %P 2:Schritt 5 = A4039 , 3: ST_CON
         IF $OUT[4039] THEN
            PREVSTEP = $APP_INT[5]
            $APP_INT[5] = 5
         ENDIF
      ;ENDFOLD
   ;ENDFOLD
   ;FOLD SCHRITT 5 -- ROB EZ1/SP1/KE1 SZ1 -- ;%{P}%MKUKATPVW,%CSTEP,%VST_NR,%P 1:SCHRITT, 2:5, 3: ROB EZ1/SP1/KE1 SZ1
      ;FOLD ;%{H}
         Case 5
      ;ENDFOLD
      ;FOLD -- Funktionstest KF Motor -- ;%{SE}%MKUKATPVW %CVW_COM %VCOMMENT %P 2:-- Funktionstest KF Motor --, 3: VW_COMMENT
      ;ENDFOLD
      ;FOLD F312 = EIN ;%{SE}%MKUKATPVW %CVW_SPS %VBOASG %P 2:F312 = EIN, 3: BOASG
         $FLAG[312] = TRUE
      ;ENDFOLD
      ;FOLD F313 = i1 > 2 ;%{SE}%MKUKATPVW %CVW_SPS %VBOCMP %P 2:F313 = i1 > 2, 3: BOCMP
         $FLAG[313] = $COUNT_I[1] > 2
      ;ENDFOLD
      ;FOLD Schritt 6 = (F313 + T7) & A4039  ;%{SE}%MKUKATPVW %CVW_SPS %VST_CON %P 2:Schritt 6 = (F313 + T7) & A4039 , 3: ST_CON
         IF ($FLAG[313] OR $TIMER_FLAG[7]) AND $OUT[4039] THEN
            PREVSTEP = $APP_INT[5]
            $APP_INT[5] = 6
         ENDIF
      ;ENDFOLD
   ;ENDFOLD
   ;FOLD SCHRITT 6 -- ROB EZ1/SP1 SZ1 -- ;%{P}%MKUKATPVW,%CSTEP,%VST_NR,%P 1:SCHRITT, 2:6, 3: ROB EZ1/SP1 SZ1
      ;FOLD ;%{H}
         Case 6
      ;ENDFOLD
      ;FOLD F312 = AUS ;%{SE}%MKUKATPVW %CVW_SPS %VBOASG %P 2:F312 = AUS, 3: BOASG
         $FLAG[312] = FALSE
      ;ENDFOLD
      ;FOLD -- KF1/KW1 Ausblasen ein -- ;%{SE}%MKUKATPVW %CVW_COM %VCOMMENT %P 2:-- KF1/KW1 Ausblasen ein --, 3: VW_COMMENT
      ;ENDFOLD
      ;FOLD A835 = (F330 + !F330 & !F331 & !F332) & !F289 ;%{SE}%MKUKATPVW %CVW_SPS %VBOASG %P 2:A835 = (F330 + !F330 & !F331 & !F332) & !F289, 3: BOASG
         $OUT[835] = ($FLAG[330] OR NOT $FLAG[330] AND NOT $FLAG[331] AND NOT $FLAG[332]) AND NOT $FLAG[289]
      ;ENDFOLD
      ;FOLD A859 = (F330 + !F330 & !F331 & !F332) & F289 ;%{SE}%MKUKATPVW %CVW_SPS %VBOASG %P 2:A859 = (F330 + !F330 & !F331 & !F332) & F289, 3: BOASG
         $OUT[859] = ($FLAG[330] OR NOT $FLAG[330] AND NOT $FLAG[331] AND NOT $FLAG[332]) AND $FLAG[289]
      ;ENDFOLD
      ;FOLD A1019 = (F330 + !F330 & !F331 & !F332) & F803 ;%{SE}%MKUKATPVW %CVW_SPS %VBOASG %P 2:A1019 = (F330 + !F330 & !F331 & !F332) & F803, 3: BOASG
         $OUT[1019] = ($FLAG[330] OR NOT $FLAG[330] AND NOT $FLAG[331] AND NOT $FLAG[332]) AND $FLAG[803]
      ;ENDFOLD
      ;FOLD Schritt 7 = A4039  ;%{SE}%MKUKATPVW %CVW_SPS %VST_CON %P 2:Schritt 7 = A4039 , 3: ST_CON
         IF $OUT[4039] THEN
            PREVSTEP = $APP_INT[5]
            $APP_INT[5] = 7
         ENDIF
      ;ENDFOLD
   ;ENDFOLD
   ;FOLD SCHRITT 7 -- ROB EZ1/SP1/KE1 SZ1 -- ;%{P}%MKUKATPVW,%CSTEP,%VST_NR,%P 1:SCHRITT, 2:7, 3: ROB EZ1/SP1/KE1 SZ1
      ;FOLD ;%{H}
         Case 7
      ;ENDFOLD
      ;FOLD -- RSK Fehlerausgabe KF1/KW1 Initiator/Motor -- ;%{SE}%MKUKATPVW %CVW_COM %VCOMMENT %P 2:-- RSK Fehlerausgabe KF1/KW1 Initiator/Motor --, 3: VW_COMMENT
      ;ENDFOLD
      ;FOLD F322 = !F313 ;%{SE}%MKUKATPVW %CVW_SPS %VBOASG %P 2:F322 = !F313, 3: BOASG
         $FLAG[322] = NOT $FLAG[313]
      ;ENDFOLD
      ;FOLD T7 ( EIN ) = STOP ;%{SE}%MKUKATPVW %CVW_SPS %VTSTOP %P 2:T7 ( EIN ) = STOP, 3: TSTOP
         VW(#SET_TIME,TRUE,7,1,0)
      ;ENDFOLD
      ;FOLD -- KF1/KW1 ein -- ;%{SE}%MKUKATPVW %CVW_COM %VCOMMENT %P 2:-- KF1/KW1 ein --, 3: VW_COMMENT
      ;ENDFOLD
      ;FOLD A834 = !F322 & !F289 ;%{SE}%MKUKATPVW %CVW_SPS %VBOASG %P 2:A834 = !F322 & !F289, 3: BOASG
         $OUT[834] = NOT $FLAG[322] AND NOT $FLAG[289]
      ;ENDFOLD
      ;FOLD A858 = !F322 & F289 ;%{SE}%MKUKATPVW %CVW_SPS %VBOASG %P 2:A858 = !F322 & F289, 3: BOASG
         $OUT[858] = NOT $FLAG[322] AND $FLAG[289]
      ;ENDFOLD
      ;FOLD A1018 = !F322 & F803 ;%{SE}%MKUKATPVW %CVW_SPS %VBOASG %P 2:A1018 = !F322 & F803, 3: BOASG
         $OUT[1018] = NOT $FLAG[322] AND $FLAG[803]
      ;ENDFOLD
      ;FOLD Schritt 8 = !F322 & A4039  ;%{SE}%MKUKATPVW %CVW_SPS %VST_CON %P 2:Schritt 8 = !F322 & A4039 , 3: ST_CON
         IF NOT $FLAG[322] AND $OUT[4039] THEN
            PREVSTEP = $APP_INT[5]
            $APP_INT[5] = 8
         ENDIF
      ;ENDFOLD
      ;FOLD Schritt 10 = F322 & A4039  ;%{SE}%MKUKATPVW %CVW_SPS %VST_CON %P 2:Schritt 10 = F322 & A4039 , 3: ST_CON
         IF $FLAG[322] AND $OUT[4039] THEN
            PREVSTEP = $APP_INT[5]
            $APP_INT[5] = 10
         ENDIF
      ;ENDFOLD
   ;ENDFOLD
   ;FOLD SCHRITT 8 -- ROB EZ1/SP1/KE1 SZ1 -- ;%{P}%MKUKATPVW,%CSTEP,%VST_NR,%P 1:SCHRITT, 2:8, 3: ROB EZ1/SP1/KE1 SZ1
      ;FOLD ;%{H}
         Case 8
      ;ENDFOLD
      ;FOLD F312 = AUS ;%{SE}%MKUKATPVW %CVW_SPS %VBOASG %P 2:F312 = AUS, 3: BOASG
         $FLAG[312] = FALSE
      ;ENDFOLD
      ;FOLD F313 = AUS ;%{SE}%MKUKATPVW %CVW_SPS %VBOASG %P 2:F313 = AUS, 3: BOASG
         $FLAG[313] = FALSE
      ;ENDFOLD
      ;FOLD -- Umdreh. KF setzen zwischenspeichern -- ;%{SE}%MKUKATPVW %CVW_COM %VCOMMENT %P 2:-- Umdreh. KF setzen zwischenspeichern --, 3: VW_COMMENT
      ;ENDFOLD
      ;FOLD F270 = F99 & F732 ;%{SE}%MKUKATPVW %CVW_SPS %VBOASG %P 2:F270 = F99 & F732, 3: BOASG
         $FLAG[270] = $FLAG[99] AND $FLAG[732]
      ;ENDFOLD
      ;FOLD i45 ( EIN ) = i4 ;%{SE}%MKUKATPVW %CVW_SPS %VARIASG %P 2:i45 ( EIN ) = i4, 3: ARIASG
         VW(#COUNTER,TRUE,45,$COUNT_I[4])
      ;ENDFOLD
      ;FOLD i4 ( F270 ) = i43 ;%{SE}%MKUKATPVW %CVW_SPS %VARIASG %P 2:i4 ( F270 ) = i43, 3: ARIASG
         VW(#COUNTER,$FLAG[270],4,$COUNT_I[43])
      ;ENDFOLD
      ;FOLD i1 ( EIN ) = 0 ;%{SE}%MKUKATPVW %CVW_SPS %VARIASG %P 2:i1 ( EIN ) = 0, 3: ARIASG
         VW(#COUNTER,TRUE,1,0)
      ;ENDFOLD
      ;FOLD -- Ueberwachungszeit EZ1/SP1/KE1 SZ1 schliessen -- ;%{SE}%MKUKATPVW %CVW_COM %VCOMMENT %P 2:-- Ueberwachungszeit EZ1/SP1/KE1 SZ1 schliessen --, 3: VW_COMMENT
      ;ENDFOLD
      ;FOLD T9 ( EIN ) = -40[1/10Sek] ;%{SE}%MKUKATPVW %CVW_SPS %VTASG %P 2:T9 ( EIN ) = -40[1/10Sek], 3: TASG
         VW(#SET_TIME,TRUE,9,0,-40)
      ;ENDFOLD
      ;FOLD -- Ueberwachungszeit KF1 -- ;%{SE}%MKUKATPVW %CVW_COM %VCOMMENT %P 2:-- Ueberwachungszeit KF1 --, 3: VW_COMMENT
      ;ENDFOLD
      ;FOLD T7 ( EIN ) = -40[1/10Sek] ;%{SE}%MKUKATPVW %CVW_SPS %VTASG %P 2:T7 ( EIN ) = -40[1/10Sek], 3: TASG
         VW(#SET_TIME,TRUE,7,0,-40)
      ;ENDFOLD
      ;FOLD Schritt 9 = A4039  ;%{SE}%MKUKATPVW %CVW_SPS %VST_CON %P 2:Schritt 9 = A4039 , 3: ST_CON
         IF $OUT[4039] THEN
            PREVSTEP = $APP_INT[5]
            $APP_INT[5] = 9
         ENDIF
      ;ENDFOLD
   ;ENDFOLD
   ;FOLD SCHRITT 9 -- ROB EZ1/SP1 SZ1 -- ;%{P}%MKUKATPVW,%CSTEP,%VST_NR,%P 1:SCHRITT, 2:9, 3: ROB EZ1/SP1 SZ1
      ;FOLD ;%{H}
         Case 9
      ;ENDFOLD
      ;FOLD -- KF1/KW1 Ausblasen ein -- ;%{SE}%MKUKATPVW %CVW_COM %VCOMMENT %P 2:-- KF1/KW1 Ausblasen ein --, 3: VW_COMMENT
      ;ENDFOLD
      ;FOLD A835 = (F330 + F331 + !F330 & !F331 & !F332) & !F289 ;%{SE}%MKUKATPVW %CVW_SPS %VBOASG %P 2:A835 = (F330 + F331 + !F330 & !F331 & !F332) & !F289, 3: BOASG
         $OUT[835] = ($FLAG[330] OR $FLAG[331] OR NOT $FLAG[330] AND NOT $FLAG[331] AND NOT $FLAG[332]) AND NOT $FLAG[289]
      ;ENDFOLD
      ;FOLD A859 = (F330 + F331 + !F330 & !F331 & !F332) & F289 ;%{SE}%MKUKATPVW %CVW_SPS %VBOASG %P 2:A859 = (F330 + F331 + !F330 & !F331 & !F332) & F289, 3: BOASG
         $OUT[859] = ($FLAG[330] OR $FLAG[331] OR NOT $FLAG[330] AND NOT $FLAG[331] AND NOT $FLAG[332]) AND $FLAG[289]
      ;ENDFOLD
      ;FOLD A1019 = (F330 + F331 + !F330 & !F331 & !F332) & F803 ;%{SE}%MKUKATPVW %CVW_SPS %VBOASG %P 2:A1019 = (F330 + F331 + !F330 & !F331 & !F332) & F803, 3: BOASG
         $OUT[1019] = ($FLAG[330] OR $FLAG[331] OR NOT $FLAG[330] AND NOT $FLAG[331] AND NOT $FLAG[332]) AND $FLAG[803]
      ;ENDFOLD
      ;FOLD -- EZ1/SP1 SZ1 schliessen -- ;%{SE}%MKUKATPVW %CVW_COM %VCOMMENT %P 2:-- EZ1/SP1 SZ1 schliessen --, 3: VW_COMMENT
      ;ENDFOLD
      ;FOLD A717 = AUS ;%{SE}%MKUKATPVW %CVW_SPS %VBOASG %P 2:A717 = AUS, 3: BOASG
         $OUT[717] = FALSE
      ;ENDFOLD
      ;FOLD A718 = EIN ;%{SE}%MKUKATPVW %CVW_SPS %VBOASG %P 2:A718 = EIN, 3: BOASG
         $OUT[718] = TRUE
      ;ENDFOLD
      ;FOLD Schritt 10 = (!E717 & E718 + T9) & A4039  ;%{SE}%MKUKATPVW %CVW_SPS %VST_CON %P 2:Schritt 10 = (!E717 & E718 + T9) & A4039 , 3: ST_CON
         IF (NOT $IN[717] AND $IN[718] OR $TIMER_FLAG[9]) AND $OUT[4039] THEN
            PREVSTEP = $APP_INT[5]
            $APP_INT[5] = 10
         ENDIF
      ;ENDFOLD
   ;ENDFOLD
   ;FOLD SCHRITT 10 -- ROB EZ1/SP1/KE1 SZ1 -- ;%{P}%MKUKATPVW,%CSTEP,%VST_NR,%P 1:SCHRITT, 2:10, 3: ROB EZ1/SP1/KE1 SZ1
      ;FOLD ;%{H}
         Case 10
      ;ENDFOLD
      ;FOLD T9 ( EIN ) = STOP ;%{SE}%MKUKATPVW %CVW_SPS %VTSTOP %P 2:T9 ( EIN ) = STOP, 3: TSTOP
         VW(#SET_TIME,TRUE,9,1,0)
      ;ENDFOLD
      ;FOLD -- RSK Fehlerausgabe Kraftaufbau -- ;%{SE}%MKUKATPVW %CVW_COM %VCOMMENT %P 2:-- RSK Fehlerausgabe Kraftaufbau --, 3: VW_COMMENT
      ;ENDFOLD
      ;FOLD F325 = T9 ;%{SE}%MKUKATPVW %CVW_SPS %VBOASG %P 2:F325 = T9, 3: BOASG
         $FLAG[325] = $TIMER_FLAG[9]
      ;ENDFOLD
      ;FOLD -- KF1/KW1 abschalten bei Fehler -- ;%{SE}%MKUKATPVW %CVW_COM %VCOMMENT %P 2:-- KF1/KW1 abschalten bei Fehler --, 3: VW_COMMENT
      ;ENDFOLD
      ;FOLD A834 = !T7 & !T9 & !F289 ;%{SE}%MKUKATPVW %CVW_SPS %VBOASG %P 2:A834 = !T7 & !T9 & !F289, 3: BOASG
         $OUT[834] = NOT $TIMER_FLAG[7] AND NOT $TIMER_FLAG[9] AND NOT $FLAG[289]
      ;ENDFOLD
      ;FOLD A858 = !T7 & !T9 & F289 ;%{SE}%MKUKATPVW %CVW_SPS %VBOASG %P 2:A858 = !T7 & !T9 & F289, 3: BOASG
         $OUT[858] = NOT $TIMER_FLAG[7] AND NOT $TIMER_FLAG[9] AND $FLAG[289]
      ;ENDFOLD
      ;FOLD A1018 = !T7 & !T9 & F803 ;%{SE}%MKUKATPVW %CVW_SPS %VBOASG %P 2:A1018 = !T7 & !T9 & F803, 3: BOASG
         $OUT[1018] = NOT $TIMER_FLAG[7] AND NOT $TIMER_FLAG[9] AND $FLAG[803]
      ;ENDFOLD
      ;FOLD -- KF1/KW1 Ausblasen -- ;%{SE}%MKUKATPVW %CVW_COM %VCOMMENT %P 2:-- KF1/KW1 Ausblasen --, 3: VW_COMMENT
      ;ENDFOLD
      ;FOLD A835 = (F330 + F331 + !F330 & !F331 & !F332) & !T9 & !F289 ;%{SE}%MKUKATPVW %CVW_SPS %VBOASG %P 2:A835 = (F330 + F331 + !F330 & !F331 & !F332) & !T9 & !F289, 3: BOASG
         $OUT[835] = ($FLAG[330] OR $FLAG[331] OR NOT $FLAG[330] AND NOT $FLAG[331] AND NOT $FLAG[332]) AND NOT $TIMER_FLAG[9] AND NOT $FLAG[289]
      ;ENDFOLD
      ;FOLD A859 = (F330 + F331 + !F330 & !F331 & !F332) & !T9 & F289 ;%{SE}%MKUKATPVW %CVW_SPS %VBOASG %P 2:A859 = (F330 + F331 + !F330 & !F331 & !F332) & !T9 & F289, 3: BOASG
         $OUT[859] = ($FLAG[330] OR $FLAG[331] OR NOT $FLAG[330] AND NOT $FLAG[331] AND NOT $FLAG[332]) AND NOT $TIMER_FLAG[9] AND $FLAG[289]
      ;ENDFOLD
      ;FOLD A1019 = (F330 + F331 + !F330 & !F331 & !F332) & !T9 & F803 ;%{SE}%MKUKATPVW %CVW_SPS %VBOASG %P 2:A1019 = (F330 + F331 + !F330 & !F331 & !F332) & !T9 & F803, 3: BOASG
         $OUT[1019] = ($FLAG[330] OR $FLAG[331] OR NOT $FLAG[330] AND NOT $FLAG[331] AND NOT $FLAG[332]) AND NOT $TIMER_FLAG[9] AND $FLAG[803]
      ;ENDFOLD
      ;FOLD -- Warte Fraesen fertig oder Timeout -- ;%{SE}%MKUKATPVW %CVW_COM %VCOMMENT %P 2:-- Warte Fraesen fertig oder Timeout --, 3: VW_COMMENT
      ;ENDFOLD
      ;FOLD Schritt 11 = (F79 & F98 + F78 & F94 & !F287 + F78 & F96 & F287 + T7 + T9) & A4039  ;%{SE}%MKUKATPVW %CVW_SPS %VST_CON %P 2:Schritt 11 = (F79 & F98 + F78 & F94 & !F287 + F78 & F96 & F287 + T7 + T9) & A4039 , 3: ST_CON
         IF ($FLAG[79] AND $FLAG[98] OR $FLAG[78] AND $FLAG[94] AND NOT $FLAG[287] OR $FLAG[78] AND $FLAG[96] AND $FLAG[287] OR $TIMER_FLAG[7] OR $TIMER_FLAG[9]) AND $OUT[4039] THEN
            PREVSTEP = $APP_INT[5]
            $APP_INT[5] = 11
         ENDIF
      ;ENDFOLD
   ;ENDFOLD
   ;FOLD SCHRITT 11 -- ROB EZ1/SP1/KE1 SZ1 -- ;%{P}%MKUKATPVW,%CSTEP,%VST_NR,%P 1:SCHRITT, 2:11, 3: ROB EZ1/SP1/KE1 SZ1
      ;FOLD ;%{H}
         Case 11
      ;ENDFOLD
      ;FOLD -- Hilfsflag SK Programmwechsel -- ;%{SE}%MKUKATPVW %CVW_COM %VCOMMENT %P 2:-- Hilfsflag SK Programmwechsel --, 3: VW_COMMENT
      ;ENDFOLD
      ;FOLD F334 = AUS ;%{SE}%MKUKATPVW %CVW_SPS %VBOASG %P 2:F334 = AUS, 3: BOASG
         $FLAG[334] = FALSE
      ;ENDFOLD
      ;FOLD t7 ( EIN ) = STOP ;%{SE}%MKUKATPVW %CVW_SPS %VTSTOP %P 2:t7 ( EIN ) = STOP, 3: TSTOP
         VW(#SET_TIME,TRUE,7,1,0)
      ;ENDFOLD
      ;FOLD -- EZ1/SP1 SZ1 oeffnen -- ;%{SE}%MKUKATPVW %CVW_COM %VCOMMENT %P 2:-- EZ1/SP1 SZ1 oeffnen --, 3: VW_COMMENT
      ;ENDFOLD
      ;FOLD A719 = AUS ;%{SE}%MKUKATPVW %CVW_SPS %VBOASG %P 2:A719 = AUS, 3: BOASG
         $OUT[719] = FALSE
      ;ENDFOLD
      ;FOLD A718 = AUS ;%{SE}%MKUKATPVW %CVW_SPS %VBOASG %P 2:A718 = AUS, 3: BOASG
         $OUT[718] = FALSE
      ;ENDFOLD
      ;FOLD A717 = EIN ;%{SE}%MKUKATPVW %CVW_SPS %VBOASG %P 2:A717 = EIN, 3: BOASG
         $OUT[717] = TRUE
      ;ENDFOLD
      ;FOLD -- KF1/KW1 Ausblasen -- ;%{SE}%MKUKATPVW %CVW_COM %VCOMMENT %P 2:-- KF1/KW1 Ausblasen --, 3: VW_COMMENT
      ;ENDFOLD
      ;FOLD A835 = (F330 + F331 + F332 + !F330 & !F331 & !F332) & !F289 ;%{SE}%MKUKATPVW %CVW_SPS %VBOASG %P 2:A835 = (F330 + F331 + F332 + !F330 & !F331 & !F332) & !F289, 3: BOASG
         $OUT[835] = ($FLAG[330] OR $FLAG[331] OR $FLAG[332] OR NOT $FLAG[330] AND NOT $FLAG[331] AND NOT $FLAG[332]) AND NOT $FLAG[289]
      ;ENDFOLD
      ;FOLD A859 = (F330 + F331 + F332 + !F330 & !F331 & !F332) & F289 ;%{SE}%MKUKATPVW %CVW_SPS %VBOASG %P 2:A859 = (F330 + F331 + F332 + !F330 & !F331 & !F332) & F289, 3: BOASG
         $OUT[859] = ($FLAG[330] OR $FLAG[331] OR $FLAG[332] OR NOT $FLAG[330] AND NOT $FLAG[331] AND NOT $FLAG[332]) AND $FLAG[289]
      ;ENDFOLD
      ;FOLD A1019 = (F330 + F331 + F332 + !F330 & !F331 & !F332) & F803 ;%{SE}%MKUKATPVW %CVW_SPS %VBOASG %P 2:A1019 = (F330 + F331 + F332 + !F330 & !F331 & !F332) & F803, 3: BOASG
         $OUT[1019] = ($FLAG[330] OR $FLAG[331] OR $FLAG[332] OR NOT $FLAG[330] AND NOT $FLAG[331] AND NOT $FLAG[332]) AND $FLAG[803]
      ;ENDFOLD
      ;FOLD -- KF Ausblasen Ausschaltverzoegerung starten -- ;%{SE}%MKUKATPVW %CVW_COM %VCOMMENT %P 2:-- KF Ausblasen Ausschaltverzoegerung starten --, 3: VW_COMMENT
      ;ENDFOLD
      ;FOLD F736 = EIN ;%{SE}%MKUKATPVW %CVW_SPS %VBOASG %P 2:F736 = EIN, 3: BOASG
         $FLAG[736] = TRUE
      ;ENDFOLD
      ;FOLD -- RSK Sammelstoerung -- ;%{SE}%MKUKATPVW %CVW_COM %VCOMMENT %P 2:-- RSK Sammelstoerung --, 3: VW_COMMENT
      ;ENDFOLD
      ;FOLD F329 = T7 + T9 ;%{SE}%MKUKATPVW %CVW_SPS %VBOASG %P 2:F329 = T7 + T9, 3: BOASG
         $FLAG[329] = $TIMER_FLAG[7] OR $TIMER_FLAG[9]
      ;ENDFOLD
      ;FOLD -- Hilfsflag Startfraesen -- ;%{SE}%MKUKATPVW %CVW_COM %VCOMMENT %P 2:-- Hilfsflag Startfraesen --, 3: VW_COMMENT
      ;ENDFOLD
      ;FOLD F96 = (F96 & F78 + F98 & F79) & F287 ;%{SE}%MKUKATPVW %CVW_SPS %VBOASG %P 2:F96 = (F96 & F78 + F98 & F79) & F287, 3: BOASG
         $FLAG[96] = ($FLAG[96] AND $FLAG[78] OR $FLAG[98] AND $FLAG[79]) AND $FLAG[287]
      ;ENDFOLD
      ;FOLD F98 = !F130 & F98 + F130 & F287 & F98 ;%{SE}%MKUKATPVW %CVW_SPS %VBOASG %P 2:F98 = !F130 & F98 + F130 & F287 & F98, 3: BOASG
         $FLAG[98] = NOT $FLAG[130] AND $FLAG[98] OR $FLAG[130] AND $FLAG[287] AND $FLAG[98]
      ;ENDFOLD
      ;FOLD F287 = F78 + F79 & F130 ;%{SE}%MKUKATPVW %CVW_SPS %VBOASG %P 2:F287 = F78 + F79 & F130, 3: BOASG
         $FLAG[287] = $FLAG[78] OR $FLAG[79] AND $FLAG[130]
      ;ENDFOLD
      ;FOLD -- Neues Fraesprogramm und Zaehler ruecksetzen -- ;%{SE}%MKUKATPVW %CVW_COM %VCOMMENT %P 2:-- Neues Fraesprogramm und Zaehler ruecksetzen --, 3: VW_COMMENT
      ;ENDFOLD
      ;FOLD F270 = F96 & F732 ;%{SE}%MKUKATPVW %CVW_SPS %VBOASG %P 2:F270 = F96 & F732, 3: BOASG
         $FLAG[270] = $FLAG[96] AND $FLAG[732]
      ;ENDFOLD
      ;FOLD bin3 ( F732 ) = 36 ;%{SE}%MKUKATPVW %CVW_SPS %VARIASG %P 2:bin3 ( F732 ) = 36, 3: ARIASG
         VW(#BINOUT,$FLAG[732],3,36)
      ;ENDFOLD
      ;FOLD i4 ( F270 ) = i45 ;%{SE}%MKUKATPVW %CVW_SPS %VARIASG %P 2:i4 ( F270 ) = i45, 3: ARIASG
         VW(#COUNTER,$FLAG[270],4,$COUNT_I[45])
      ;ENDFOLD
      ;FOLD -- Wiederholung beim Startfraesen -- ;%{SE}%MKUKATPVW %CVW_COM %VCOMMENT %P 2:-- Wiederholung beim Startfraesen --, 3: VW_COMMENT
      ;ENDFOLD
      ;FOLD Schritt 8 = E717 & !E718 & (F78 & !F96 + F79 & F130 & !F96) & !F329 & A4039  ;%{SE}%MKUKATPVW %CVW_SPS %VST_CON %P 2:Schritt 8 = E717 & !E718 & (F78 & !F96 + F79 & F130 & !F96) & !F329 & A4039 , 3: ST_CON
         IF $IN[717] AND NOT $IN[718] AND ($FLAG[78] AND NOT $FLAG[96] OR $FLAG[79] AND $FLAG[130] AND NOT $FLAG[96]) AND NOT $FLAG[329] AND $OUT[4039] THEN
            PREVSTEP = $APP_INT[5]
            $APP_INT[5] = 8
         ENDIF
      ;ENDFOLD
      ;FOLD -- Weiter wenn Fraesen fertig -- ;%{SE}%MKUKATPVW %CVW_COM %VCOMMENT %P 2:-- Weiter wenn Fraesen fertig --, 3: VW_COMMENT
      ;ENDFOLD
      ;FOLD Schritt 12 = E717 & !E718 & (F79 & F98 & (!F130 + F96) + F78 & F96 + F329) & A4039  ;%{SE}%MKUKATPVW %CVW_SPS %VST_CON %P 2:Schritt 12 = E717 & !E718 & (F79 & F98 & (!F130 + F96) + F78 & F96 + F329) & A4039 , 3: ST_CON
         IF $IN[717] AND NOT $IN[718] AND ($FLAG[79] AND $FLAG[98] AND (NOT $FLAG[130] OR $FLAG[96]) OR $FLAG[78] AND $FLAG[96] OR $FLAG[329]) AND $OUT[4039] THEN
            PREVSTEP = $APP_INT[5]
            $APP_INT[5] = 12
         ENDIF
      ;ENDFOLD
      ;FOLD -- Weiter bei Fehler -- ;%{SE}%MKUKATPVW %CVW_COM %VCOMMENT %P 2:-- Weiter bei Fehler --, 3: VW_COMMENT
      ;ENDFOLD
      ;FOLD Schritt 14 = F325 & (E26 + E27) & A4039  ;%{SE}%MKUKATPVW %CVW_SPS %VST_CON %P 2:Schritt 14 = F325 & (E26 + E27) & A4039 , 3: ST_CON
         IF $FLAG[325] AND ($IN[26] OR $IN[27]) AND $OUT[4039] THEN
            PREVSTEP = $APP_INT[5]
            $APP_INT[5] = 14
         ENDIF
      ;ENDFOLD
   ;ENDFOLD
   ;FOLD SCHRITT 12 -- ROB EZ1/SP1/KE1 SZ1 -- ;%{P}%MKUKATPVW,%CSTEP,%VST_NR,%P 1:SCHRITT, 2:12, 3: ROB EZ1/SP1/KE1 SZ1
      ;FOLD ;%{H}
         Case 12
      ;ENDFOLD
      ;FOLD F270 = AUS ;%{SE}%MKUKATPVW %CVW_SPS %VBOASG %P 2:F270 = AUS, 3: BOASG
         $FLAG[270] = FALSE
      ;ENDFOLD
      ;FOLD A717 = AUS ;%{SE}%MKUKATPVW %CVW_SPS %VBOASG %P 2:A717 = AUS, 3: BOASG
         $OUT[717] = FALSE
      ;ENDFOLD
      ;FOLD -- KF1/KW1 abschalten -- ;%{SE}%MKUKATPVW %CVW_COM %VCOMMENT %P 2:-- KF1/KW1 abschalten --, 3: VW_COMMENT
      ;ENDFOLD
      ;FOLD A834 = AUS ;%{SE}%MKUKATPVW %CVW_SPS %VBOASG %P 2:A834 = AUS, 3: BOASG
         $OUT[834] = FALSE
      ;ENDFOLD
      ;FOLD A858 = AUS ;%{SE}%MKUKATPVW %CVW_SPS %VBOASG %P 2:A858 = AUS, 3: BOASG
         $OUT[858] = FALSE
      ;ENDFOLD
      ;FOLD A1018 = AUS ;%{SE}%MKUKATPVW %CVW_SPS %VBOASG %P 2:A1018 = AUS, 3: BOASG
         $OUT[1018] = FALSE
      ;ENDFOLD
      ;FOLD bin3 ( !F329 ) = 1 ;%{SE}%MKUKATPVW %CVW_SPS %VARIASG %P 2:bin3 ( !F329 ) = 1, 3: ARIASG
         VW(#BINOUT,NOT $FLAG[329],3,1)
      ;ENDFOLD
      ;FOLD -- Wartezeit Programmwechsel SK -- ;%{SE}%MKUKATPVW %CVW_COM %VCOMMENT %P 2:-- Wartezeit Programmwechsel SK --, 3: VW_COMMENT
      ;ENDFOLD
      ;FOLD T8 ( !F334 ) = -2[1/10Sek] ;%{SE}%MKUKATPVW %CVW_SPS %VTASG %P 2:T8 ( !F334 ) = -2[1/10Sek], 3: TASG
         VW(#SET_TIME,NOT $FLAG[334],8,0,-2)
      ;ENDFOLD
      ;FOLD -- Hilfsflag SK Programmwechsel -- ;%{SE}%MKUKATPVW %CVW_COM %VCOMMENT %P 2:-- Hilfsflag SK Programmwechsel --, 3: VW_COMMENT
      ;ENDFOLD
      ;FOLD F334 = EIN ;%{SE}%MKUKATPVW %CVW_SPS %VBOASG %P 2:F334 = EIN, 3: BOASG
         $FLAG[334] = TRUE
      ;ENDFOLD
      ;FOLD Schritt 13 = T8 & A4039  ;%{SE}%MKUKATPVW %CVW_SPS %VST_CON %P 2:Schritt 13 = T8 & A4039 , 3: ST_CON
         IF $TIMER_FLAG[8] AND $OUT[4039] THEN
            PREVSTEP = $APP_INT[5]
            $APP_INT[5] = 13
         ENDIF
      ;ENDFOLD
   ;ENDFOLD
   ;FOLD SCHRITT 13 -- ROB EZ1/SP1/KE1 SZ1 -- ;%{P}%MKUKATPVW,%CSTEP,%VST_NR,%P 1:SCHRITT, 2:13, 3: ROB EZ1/SP1/KE1 SZ1
      ;FOLD ;%{H}
         Case 13
      ;ENDFOLD
      ;FOLD -- Hilfsflag SK Programmwechsel -- ;%{SE}%MKUKATPVW %CVW_COM %VCOMMENT %P 2:-- Hilfsflag SK Programmwechsel --, 3: VW_COMMENT
      ;ENDFOLD
      ;FOLD F334 = AUS ;%{SE}%MKUKATPVW %CVW_SPS %VBOASG %P 2:F334 = AUS, 3: BOASG
         $FLAG[334] = FALSE
      ;ENDFOLD
      ;FOLD -- Quitt. Fraesen SK1 -- ;%{SE}%MKUKATPVW %CVW_COM %VCOMMENT %P 2:-- Quitt. Fraesen SK1 --, 3: VW_COMMENT
      ;ENDFOLD
      ;FOLD A786 = (!F329 & !F322 & !F830) + (F830 & A786) ;%{SE}%MKUKATPVW %CVW_SPS %VBOASG %P 2:A786 = (!F329 & !F322 & !F830) + (F830 & A786), 3: BOASG
         $OUT[786] = (NOT $FLAG[329] AND NOT $FLAG[322] AND NOT $FLAG[830]) OR ($FLAG[830] AND $OUT[786])
      ;ENDFOLD
      ;FOLD A722 = (!F329 & !F322 & F830) + (!F830 & A722) ;%{SE}%MKUKATPVW %CVW_SPS %VBOASG %P 2:A722 = (!F329 & !F322 & F830) + (!F830 & A722), 3: BOASG
         $OUT[722] = (NOT $FLAG[329] AND NOT $FLAG[322] AND $FLAG[830]) OR (NOT $FLAG[830] AND $OUT[722])
      ;ENDFOLD
      ;FOLD Schritt 14 = (!F830 & !E786 & E787 & !E788 + F830 & !E722 & E724 & !E723 + F329) & A4039  ;%{SE}%MKUKATPVW %CVW_SPS %VST_CON %P 2:Schritt 14 = (!F830 & !E786 & E787 & !E788 + F830 & !E722 & E724 & !E723 + F329) & A4039 , 3: ST_CON
         IF (NOT $FLAG[830] AND NOT $IN[786] AND $IN[787] AND NOT $IN[788] OR $FLAG[830] AND NOT $IN[722] AND $IN[724] AND NOT $IN[723] OR $FLAG[329]) AND $OUT[4039] THEN
            PREVSTEP = $APP_INT[5]
            $APP_INT[5] = 14
         ENDIF
      ;ENDFOLD
   ;ENDFOLD
   ;FOLD SCHRITT 14 -- ROB EZ1/SP1/KE1 SZ1 # Ende-- ;%{P}%MKUKATPVW,%CSTEP,%VST_NR,%P 1:SCHRITT, 2:14, 3: ROB EZ1/SP1/KE1 SZ1 # Ende
      ;FOLD ;%{H}
         Case 14
      ;ENDFOLD
      ;FOLD F270 = AUS ;%{SE}%MKUKATPVW %CVW_SPS %VBOASG %P 2:F270 = AUS, 3: BOASG
         $FLAG[270] = FALSE
      ;ENDFOLD
      ;FOLD -- KF1/KW1 Ausblasen -- ;%{SE}%MKUKATPVW %CVW_COM %VCOMMENT %P 2:-- KF1/KW1 Ausblasen --, 3: VW_COMMENT
      ;ENDFOLD
      ;FOLD A835 = (F330 + F331 + F332) & F736 ;%{SE}%MKUKATPVW %CVW_SPS %VBOASG %P 2:A835 = (F330 + F331 + F332) & F736, 3: BOASG
         $OUT[835] = ($FLAG[330] OR $FLAG[331] OR $FLAG[332]) AND $FLAG[736]
      ;ENDFOLD
      ;FOLD A859 = (F330 + F331 + F332) & F736 & F289 ;%{SE}%MKUKATPVW %CVW_SPS %VBOASG %P 2:A859 = (F330 + F331 + F332) & F736 & F289, 3: BOASG
         $OUT[859] = ($FLAG[330] OR $FLAG[331] OR $FLAG[332]) AND $FLAG[736] AND $FLAG[289]
      ;ENDFOLD
      ;FOLD A1019 = (F330 + F331 + F332) & F736 & F803 ;%{SE}%MKUKATPVW %CVW_SPS %VBOASG %P 2:A1019 = (F330 + F331 + F332) & F736 & F803, 3: BOASG
         $OUT[1019] = ($FLAG[330] OR $FLAG[331] OR $FLAG[332]) AND $FLAG[736] AND $FLAG[803]
      ;ENDFOLD
      ;FOLD F91 = (!E786 & E787 & !E788 & !F830 + !E722 & E724 & !E723 & F830) & !F322 & !F325 & !F329 ;%{SE}%MKUKATPVW %CVW_SPS %VBOASG %P 2:F91 = (!E786 & E787 & !E788 & !F830 + !E722 & E724 & !E723 & F830) & !F322 & !F325 & !F329, 3: BOASG
         $FLAG[91] = (NOT $IN[786] AND $IN[787] AND NOT $IN[788] AND NOT $FLAG[830] OR NOT $IN[722] AND $IN[724] AND NOT $IN[723] AND $FLAG[830]) AND NOT $FLAG[322] AND NOT $FLAG[325] AND NOT $FLAG[329]
      ;ENDFOLD
      ;FOLD Schritt 3 = (F322 + F325 + F329) & (E26 + E27) & A4039  ;%{SE}%MKUKATPVW %CVW_SPS %VST_CON %P 2:Schritt 3 = (F322 + F325 + F329) & (E26 + E27) & A4039 , 3: ST_CON
         IF ($FLAG[322] OR $FLAG[325] OR $FLAG[329]) AND ($IN[26] OR $IN[27]) AND $OUT[4039] THEN
            PREVSTEP = $APP_INT[5]
            $APP_INT[5] = 3
         ENDIF
      ;ENDFOLD
      ;FOLD Schritt 1 = F91 & !F322 & !F325 & !F329 & A4039  ;%{SE}%MKUKATPVW %CVW_SPS %VST_CON %P 2:Schritt 1 = F91 & !F322 & !F325 & !F329 & A4039 , 3: ST_CON
         IF $FLAG[91] AND NOT $FLAG[322] AND NOT $FLAG[325] AND NOT $FLAG[329] AND $OUT[4039] THEN
            PREVSTEP = $APP_INT[5]
            $APP_INT[5] = 1
         ENDIF
      ;ENDFOLD
   ;ENDFOLD
   ;FOLD SCHRITT 15 -- ROB EZ1/SP1/KE1 SZ2 # Start-- ;%{P}%MKUKATPVW,%CSTEP,%VST_NR,%P 1:SCHRITT, 2:15, 3: ROB EZ1/SP1/KE1 SZ2 # Start
      ;FOLD ;%{H}
         Case 15
      ;ENDFOLD
      ;FOLD -- RSK gestartet -- ;%{SE}%MKUKATPVW %CVW_COM %VCOMMENT %P 2:-- RSK gestartet --, 3: VW_COMMENT
      ;ENDFOLD
      ;FOLD F321 = AUS ;%{SE}%MKUKATPVW %CVW_SPS %VBOASG %P 2:F321 = AUS, 3: BOASG
         $FLAG[321] = FALSE
      ;ENDFOLD
      ;FOLD F322 = AUS ;%{SE}%MKUKATPVW %CVW_SPS %VBOASG %P 2:F322 = AUS, 3: BOASG
         $FLAG[322] = FALSE
      ;ENDFOLD
      ;FOLD F323 = AUS ;%{SE}%MKUKATPVW %CVW_SPS %VBOASG %P 2:F323 = AUS, 3: BOASG
         $FLAG[323] = FALSE
      ;ENDFOLD
      ;FOLD F324 = AUS ;%{SE}%MKUKATPVW %CVW_SPS %VBOASG %P 2:F324 = AUS, 3: BOASG
         $FLAG[324] = FALSE
      ;ENDFOLD
      ;FOLD F325 = AUS ;%{SE}%MKUKATPVW %CVW_SPS %VBOASG %P 2:F325 = AUS, 3: BOASG
         $FLAG[325] = FALSE
      ;ENDFOLD
      ;FOLD F327 = AUS ;%{SE}%MKUKATPVW %CVW_SPS %VBOASG %P 2:F327 = AUS, 3: BOASG
         $FLAG[327] = FALSE
      ;ENDFOLD
      ;FOLD F329 = AUS ;%{SE}%MKUKATPVW %CVW_SPS %VBOASG %P 2:F329 = AUS, 3: BOASG
         $FLAG[329] = FALSE
      ;ENDFOLD
      ;FOLD -- EZ1/SP1/KE1 SZ2 Zaehler -- ;%{SE}%MKUKATPVW %CVW_COM %VCOMMENT %P 2:-- EZ1/SP1/KE1 SZ2 Zaehler --, 3: VW_COMMENT
      ;ENDFOLD
      ;FOLD F100 = AUS ;%{SE}%MKUKATPVW %CVW_SPS %VBOASG %P 2:F100 = AUS, 3: BOASG
         $FLAG[100] = FALSE
      ;ENDFOLD
      ;FOLD F101 = AUS ;%{SE}%MKUKATPVW %CVW_SPS %VBOASG %P 2:F101 = AUS, 3: BOASG
         $FLAG[101] = FALSE
      ;ENDFOLD
      ;FOLD F102 = AUS ;%{SE}%MKUKATPVW %CVW_SPS %VBOASG %P 2:F102 = AUS, 3: BOASG
         $FLAG[102] = FALSE
      ;ENDFOLD
      ;FOLD F103 = AUS ;%{SE}%MKUKATPVW %CVW_SPS %VBOASG %P 2:F103 = AUS, 3: BOASG
         $FLAG[103] = FALSE
      ;ENDFOLD
      ;FOLD F104 = AUS ;%{SE}%MKUKATPVW %CVW_SPS %VBOASG %P 2:F104 = AUS, 3: BOASG
         $FLAG[104] = FALSE
      ;ENDFOLD
      ;FOLD F105 = AUS ;%{SE}%MKUKATPVW %CVW_SPS %VBOASG %P 2:F105 = AUS, 3: BOASG
         $FLAG[105] = FALSE
      ;ENDFOLD
      ;FOLD -- Hilfsflags Funktionstest KF Motor -- ;%{SE}%MKUKATPVW %CVW_COM %VCOMMENT %P 2:-- Hilfsflags Funktionstest KF Motor --, 3: VW_COMMENT
      ;ENDFOLD
      ;FOLD F312 = AUS ;%{SE}%MKUKATPVW %CVW_SPS %VBOASG %P 2:F312 = AUS, 3: BOASG
         $FLAG[312] = FALSE
      ;ENDFOLD
      ;FOLD F313 = AUS ;%{SE}%MKUKATPVW %CVW_SPS %VBOASG %P 2:F313 = AUS, 3: BOASG
         $FLAG[313] = FALSE
      ;ENDFOLD
      ;FOLD -- Rob. EZ1/SP1/KE1 SZ2 beim Fraesen -- ;%{SE}%MKUKATPVW %CVW_COM %VCOMMENT %P 2:-- Rob. EZ1/SP1/KE1 SZ2 beim Fraesen --, 3: VW_COMMENT
      ;ENDFOLD
      ;FOLD A116 = EIN ;%{SE}%MKUKATPVW %CVW_SPS %VBOASG %P 2:A116 = EIN, 3: BOASG
         $OUT[116] = TRUE
      ;ENDFOLD
      ;FOLD A130 = EIN ;%{SE}%MKUKATPVW %CVW_SPS %VBOASG %P 2:A130 = EIN, 3: BOASG
         $OUT[130] = TRUE
      ;ENDFOLD
      ;FOLD -- Quitt. Fraesen SK1/KE1 AUS -- ;%{SE}%MKUKATPVW %CVW_COM %VCOMMENT %P 2:-- Quitt. Fraesen SK1/KE1 AUS --, 3: VW_COMMENT
      ;ENDFOLD
      ;FOLD A786 = F830 & A786 ;%{SE}%MKUKATPVW %CVW_SPS %VBOASG %P 2:A786 = F830 & A786, 3: BOASG
         $OUT[786] = $FLAG[830] AND $OUT[786]
      ;ENDFOLD
      ;FOLD A722 = !F830 & A722 ;%{SE}%MKUKATPVW %CVW_SPS %VBOASG %P 2:A722 = !F830 & A722, 3: BOASG
         $OUT[722] = NOT $FLAG[830] AND $OUT[722]
      ;ENDFOLD
      ;FOLD -- Ueberwachungszeit KF1/KW1 -- ;%{SE}%MKUKATPVW %CVW_COM %VCOMMENT %P 2:-- Ueberwachungszeit KF1/KW1 --, 3: VW_COMMENT
      ;ENDFOLD
      ;FOLD t7 ( EIN ) = -30[1/10Sek] ;%{SE}%MKUKATPVW %CVW_SPS %VTASG %P 2:t7 ( EIN ) = -30[1/10Sek], 3: TASG
         VW(#SET_TIME,TRUE,7,0,-30)
      ;ENDFOLD
      ;FOLD Schritt 16 = A4039  ;%{SE}%MKUKATPVW %CVW_SPS %VST_CON %P 2:Schritt 16 = A4039 , 3: ST_CON
         IF $OUT[4039] THEN
            PREVSTEP = $APP_INT[5]
            $APP_INT[5] = 16
         ENDIF
      ;ENDFOLD
   ;ENDFOLD
   ;FOLD SCHRITT 16 -- ROB EZ1/SP1/KE1 SZ2 -- ;%{P}%MKUKATPVW,%CSTEP,%VST_NR,%P 1:SCHRITT, 2:16, 3: ROB EZ1/SP1/KE1 SZ2
      ;FOLD ;%{H}
         Case 16
      ;ENDFOLD
      ;FOLD -- KF1/KW1 einschalten -- ;%{SE}%MKUKATPVW %CVW_COM %VCOMMENT %P 2:-- KF1/KW1 einschalten --, 3: VW_COMMENT
      ;ENDFOLD
      ;FOLD i1 ( EIN ) = 0 ;%{SE}%MKUKATPVW %CVW_SPS %VARIASG %P 2:i1 ( EIN ) = 0, 3: ARIASG
         VW(#COUNTER,TRUE,1,0)
      ;ENDFOLD
      ;FOLD A834 = !F289 & !F72 & !F73 ;%{SE}%MKUKATPVW %CVW_SPS %VBOASG %P 2:A834 = !F289 & !F72 & !F73, 3: BOASG
         $OUT[834] = NOT $FLAG[289] AND NOT $FLAG[72] AND NOT $FLAG[73]
      ;ENDFOLD
      ;FOLD A858 = F289 & !F72 & !F73 ;%{SE}%MKUKATPVW %CVW_SPS %VBOASG %P 2:A858 = F289 & !F72 & !F73, 3: BOASG
         $OUT[858] = $FLAG[289] AND NOT $FLAG[72] AND NOT $FLAG[73]
      ;ENDFOLD
      ;FOLD -- KF2/KW2 einschalten -- ;%{SE}%MKUKATPVW %CVW_COM %VCOMMENT %P 2:-- KF2/KW2 einschalten --, 3: VW_COMMENT
      ;ENDFOLD
      ;FOLD A994 = !F803 & F72 ;%{SE}%MKUKATPVW %CVW_SPS %VBOASG %P 2:A994 = !F803 & F72, 3: BOASG
         $OUT[994] = NOT $FLAG[803] AND $FLAG[72]
      ;ENDFOLD
      ;FOLD A1018 = F803 & F72 ;%{SE}%MKUKATPVW %CVW_SPS %VBOASG %P 2:A1018 = F803 & F72, 3: BOASG
         $OUT[1018] = $FLAG[803] AND $FLAG[72]
      ;ENDFOLD
      ;FOLD -- KF3/KW3 einschalten -- ;%{SE}%MKUKATPVW %CVW_COM %VCOMMENT %P 2:-- KF3/KW3 einschalten --, 3: VW_COMMENT
      ;ENDFOLD
      ;FOLD A1154 = !F804 & F73 ;%{SE}%MKUKATPVW %CVW_SPS %VBOASG %P 2:A1154 = !F804 & F73, 3: BOASG
         $OUT[1154] = NOT $FLAG[804] AND $FLAG[73]
      ;ENDFOLD
      ;FOLD A1178 = F804 & F73 ;%{SE}%MKUKATPVW %CVW_SPS %VBOASG %P 2:A1178 = F804 & F73, 3: BOASG
         $OUT[1178] = $FLAG[804] AND $FLAG[73]
      ;ENDFOLD
      ;FOLD Schritt 17 = A4039  ;%{SE}%MKUKATPVW %CVW_SPS %VST_CON %P 2:Schritt 17 = A4039 , 3: ST_CON
         IF $OUT[4039] THEN
            PREVSTEP = $APP_INT[5]
            $APP_INT[5] = 17
         ENDIF
      ;ENDFOLD
   ;ENDFOLD
   ;FOLD SCHRITT 17 -- ROB EZ1/SP1/KE1 SZ2 -- ;%{P}%MKUKATPVW,%CSTEP,%VST_NR,%P 1:SCHRITT, 2:17, 3: ROB EZ1/SP1/KE1 SZ2
      ;FOLD ;%{H}
         Case 17
      ;ENDFOLD
      ;FOLD -- Funktionstest KF Motor -- ;%{SE}%MKUKATPVW %CVW_COM %VCOMMENT %P 2:-- Funktionstest KF Motor --, 3: VW_COMMENT
      ;ENDFOLD
      ;FOLD F312 = EIN ;%{SE}%MKUKATPVW %CVW_SPS %VBOASG %P 2:F312 = EIN, 3: BOASG
         $FLAG[312] = TRUE
      ;ENDFOLD
      ;FOLD F313 = i1 > 2 ;%{SE}%MKUKATPVW %CVW_SPS %VBOCMP %P 2:F313 = i1 > 2, 3: BOCMP
         $FLAG[313] = $COUNT_I[1] > 2
      ;ENDFOLD
      ;FOLD Schritt 18 = (F313 + T7) & A4039  ;%{SE}%MKUKATPVW %CVW_SPS %VST_CON %P 2:Schritt 18 = (F313 + T7) & A4039 , 3: ST_CON
         IF ($FLAG[313] OR $TIMER_FLAG[7]) AND $OUT[4039] THEN
            PREVSTEP = $APP_INT[5]
            $APP_INT[5] = 18
         ENDIF
      ;ENDFOLD
   ;ENDFOLD
   ;FOLD SCHRITT 18 -- ROB EZ1/SP1 SZ2 -- ;%{P}%MKUKATPVW,%CSTEP,%VST_NR,%P 1:SCHRITT, 2:18, 3: ROB EZ1/SP1 SZ2
      ;FOLD ;%{H}
         Case 18
      ;ENDFOLD
      ;FOLD F312 = AUS ;%{SE}%MKUKATPVW %CVW_SPS %VBOASG %P 2:F312 = AUS, 3: BOASG
         $FLAG[312] = FALSE
      ;ENDFOLD
      ;FOLD -- KF1/KW1 Ausblasen ein -- ;%{SE}%MKUKATPVW %CVW_COM %VCOMMENT %P 2:-- KF1/KW1 Ausblasen ein --, 3: VW_COMMENT
      ;ENDFOLD
      ;FOLD A835 = (F330 + !F330 & !F331 & !F332) & !F289 & !F72 & !F73 ;%{SE}%MKUKATPVW %CVW_SPS %VBOASG %P 2:A835 = (F330 + !F330 & !F331 & !F332) & !F289 & !F72 & !F73, 3: BOASG
         $OUT[835] = ($FLAG[330] OR NOT $FLAG[330] AND NOT $FLAG[331] AND NOT $FLAG[332]) AND NOT $FLAG[289] AND NOT $FLAG[72] AND NOT $FLAG[73]
      ;ENDFOLD
      ;FOLD A859 = (F330 + !F330 & !F331 & !F332) & F289 & !F72 & !F73 ;%{SE}%MKUKATPVW %CVW_SPS %VBOASG %P 2:A859 = (F330 + !F330 & !F331 & !F332) & F289 & !F72 & !F73, 3: BOASG
         $OUT[859] = ($FLAG[330] OR NOT $FLAG[330] AND NOT $FLAG[331] AND NOT $FLAG[332]) AND $FLAG[289] AND NOT $FLAG[72] AND NOT $FLAG[73]
      ;ENDFOLD
      ;FOLD -- KF2/KW2 Ausblasen ein -- ;%{SE}%MKUKATPVW %CVW_COM %VCOMMENT %P 2:-- KF2/KW2 Ausblasen ein --, 3: VW_COMMENT
      ;ENDFOLD
      ;FOLD A995 = (F330 + !F330 & !F331 & !F332) & !F803 & F72 ;%{SE}%MKUKATPVW %CVW_SPS %VBOASG %P 2:A995 = (F330 + !F330 & !F331 & !F332) & !F803 & F72, 3: BOASG
         $OUT[995] = ($FLAG[330] OR NOT $FLAG[330] AND NOT $FLAG[331] AND NOT $FLAG[332]) AND NOT $FLAG[803] AND $FLAG[72]
      ;ENDFOLD
      ;FOLD A1019 = (F330 + !F330 & !F331 & !F332) & F803 & F72 ;%{SE}%MKUKATPVW %CVW_SPS %VBOASG %P 2:A1019 = (F330 + !F330 & !F331 & !F332) & F803 & F72, 3: BOASG
         $OUT[1019] = ($FLAG[330] OR NOT $FLAG[330] AND NOT $FLAG[331] AND NOT $FLAG[332]) AND $FLAG[803] AND $FLAG[72]
      ;ENDFOLD
      ;FOLD -- KF3/KW3 Ausblasen ein -- ;%{SE}%MKUKATPVW %CVW_COM %VCOMMENT %P 2:-- KF3/KW3 Ausblasen ein --, 3: VW_COMMENT
      ;ENDFOLD
      ;FOLD A1155 = (F330 + !F330 & !F331 & !F332) & !F804 & F73 ;%{SE}%MKUKATPVW %CVW_SPS %VBOASG %P 2:A1155 = (F330 + !F330 & !F331 & !F332) & !F804 & F73, 3: BOASG
         $OUT[1155] = ($FLAG[330] OR NOT $FLAG[330] AND NOT $FLAG[331] AND NOT $FLAG[332]) AND NOT $FLAG[804] AND $FLAG[73]
      ;ENDFOLD
      ;FOLD A1179 = (F330 + !F330 & !F331 & !F332) & F804 & F73 ;%{SE}%MKUKATPVW %CVW_SPS %VBOASG %P 2:A1179 = (F330 + !F330 & !F331 & !F332) & F804 & F73, 3: BOASG
         $OUT[1179] = ($FLAG[330] OR NOT $FLAG[330] AND NOT $FLAG[331] AND NOT $FLAG[332]) AND $FLAG[804] AND $FLAG[73]
      ;ENDFOLD
      ;FOLD Schritt 19 = A4039  ;%{SE}%MKUKATPVW %CVW_SPS %VST_CON %P 2:Schritt 19 = A4039 , 3: ST_CON
         IF $OUT[4039] THEN
            PREVSTEP = $APP_INT[5]
            $APP_INT[5] = 19
         ENDIF
      ;ENDFOLD
   ;ENDFOLD
   ;FOLD SCHRITT 19 -- ROB EZ1/SP1 SZ2 -- ;%{P}%MKUKATPVW,%CSTEP,%VST_NR,%P 1:SCHRITT, 2:19, 3: ROB EZ1/SP1 SZ2
      ;FOLD ;%{H}
         Case 19
      ;ENDFOLD
      ;FOLD -- RSK Fehlerausgabe KF1/KW1 Initiator/Motor -- ;%{SE}%MKUKATPVW %CVW_COM %VCOMMENT %P 2:-- RSK Fehlerausgabe KF1/KW1 Initiator/Motor --, 3: VW_COMMENT
      ;ENDFOLD
      ;FOLD F322 = !F313 ;%{SE}%MKUKATPVW %CVW_SPS %VBOASG %P 2:F322 = !F313, 3: BOASG
         $FLAG[322] = NOT $FLAG[313]
      ;ENDFOLD
      ;FOLD T7 ( EIN ) = STOP ;%{SE}%MKUKATPVW %CVW_SPS %VTSTOP %P 2:T7 ( EIN ) = STOP, 3: TSTOP
         VW(#SET_TIME,TRUE,7,1,0)
      ;ENDFOLD
      ;FOLD -- KF1/KW1 ein -- ;%{SE}%MKUKATPVW %CVW_COM %VCOMMENT %P 2:-- KF1/KW1 ein --, 3: VW_COMMENT
      ;ENDFOLD
      ;FOLD A834 = !F322 & !F289 & !F72 & !F73 ;%{SE}%MKUKATPVW %CVW_SPS %VBOASG %P 2:A834 = !F322 & !F289 & !F72 & !F73, 3: BOASG
         $OUT[834] = NOT $FLAG[322] AND NOT $FLAG[289] AND NOT $FLAG[72] AND NOT $FLAG[73]
      ;ENDFOLD
      ;FOLD A858 = !F322 & F289 & !F72 & !F73 ;%{SE}%MKUKATPVW %CVW_SPS %VBOASG %P 2:A858 = !F322 & F289 & !F72 & !F73, 3: BOASG
         $OUT[858] = NOT $FLAG[322] AND $FLAG[289] AND NOT $FLAG[72] AND NOT $FLAG[73]
      ;ENDFOLD
      ;FOLD -- KF2/KW2 ein -- ;%{SE}%MKUKATPVW %CVW_COM %VCOMMENT %P 2:-- KF2/KW2 ein --, 3: VW_COMMENT
      ;ENDFOLD
      ;FOLD A994 = !F322 & !F803 & F72 ;%{SE}%MKUKATPVW %CVW_SPS %VBOASG %P 2:A994 = !F322 & !F803 & F72, 3: BOASG
         $OUT[994] = NOT $FLAG[322] AND NOT $FLAG[803] AND $FLAG[72]
      ;ENDFOLD
      ;FOLD A1018 = !F322 & F803 & F72 ;%{SE}%MKUKATPVW %CVW_SPS %VBOASG %P 2:A1018 = !F322 & F803 & F72, 3: BOASG
         $OUT[1018] = NOT $FLAG[322] AND $FLAG[803] AND $FLAG[72]
      ;ENDFOLD
      ;FOLD -- KF3/KW3 ein -- ;%{SE}%MKUKATPVW %CVW_COM %VCOMMENT %P 2:-- KF3/KW3 ein --, 3: VW_COMMENT
      ;ENDFOLD
      ;FOLD A1154 = !F322 & !F804 & F73 ;%{SE}%MKUKATPVW %CVW_SPS %VBOASG %P 2:A1154 = !F322 & !F804 & F73, 3: BOASG
         $OUT[1154] = NOT $FLAG[322] AND NOT $FLAG[804] AND $FLAG[73]
      ;ENDFOLD
      ;FOLD A1178 = !F322 & F804 & F73 ;%{SE}%MKUKATPVW %CVW_SPS %VBOASG %P 2:A1178 = !F322 & F804 & F73, 3: BOASG
         $OUT[1178] = NOT $FLAG[322] AND $FLAG[804] AND $FLAG[73]
      ;ENDFOLD
      ;FOLD Schritt 20 = !F322 & A4039  ;%{SE}%MKUKATPVW %CVW_SPS %VST_CON %P 2:Schritt 20 = !F322 & A4039 , 3: ST_CON
         IF NOT $FLAG[322] AND $OUT[4039] THEN
            PREVSTEP = $APP_INT[5]
            $APP_INT[5] = 20
         ENDIF
      ;ENDFOLD
      ;FOLD Schritt 22 = F322 & A4039  ;%{SE}%MKUKATPVW %CVW_SPS %VST_CON %P 2:Schritt 22 = F322 & A4039 , 3: ST_CON
         IF $FLAG[322] AND $OUT[4039] THEN
            PREVSTEP = $APP_INT[5]
            $APP_INT[5] = 22
         ENDIF
      ;ENDFOLD
   ;ENDFOLD
   ;FOLD SCHRITT 20 -- ROB EZ1/SP1/KE1 SZ2 -- ;%{P}%MKUKATPVW,%CSTEP,%VST_NR,%P 1:SCHRITT, 2:20, 3: ROB EZ1/SP1/KE1 SZ2
      ;FOLD ;%{H}
         Case 20
      ;ENDFOLD
      ;FOLD F312 = AUS ;%{SE}%MKUKATPVW %CVW_SPS %VBOASG %P 2:F312 = AUS, 3: BOASG
         $FLAG[312] = FALSE
      ;ENDFOLD
      ;FOLD F313 = AUS ;%{SE}%MKUKATPVW %CVW_SPS %VBOASG %P 2:F313 = AUS, 3: BOASG
         $FLAG[313] = FALSE
      ;ENDFOLD
      ;FOLD -- Umdreh. KF setzen -- ;%{SE}%MKUKATPVW %CVW_COM %VCOMMENT %P 2:-- Umdreh. KF setzen --, 3: VW_COMMENT
      ;ENDFOLD
      ;FOLD F270 = F105 & F732 ;%{SE}%MKUKATPVW %CVW_SPS %VBOASG %P 2:F270 = F105 & F732, 3: BOASG
         $FLAG[270] = $FLAG[105] AND $FLAG[732]
      ;ENDFOLD
      ;FOLD i45 ( EIN ) = i10 ;%{SE}%MKUKATPVW %CVW_SPS %VARIASG %P 2:i45 ( EIN ) = i10, 3: ARIASG
         VW(#COUNTER,TRUE,45,$COUNT_I[10])
      ;ENDFOLD
      ;FOLD i10 ( F270 ) = i43 ;%{SE}%MKUKATPVW %CVW_SPS %VARIASG %P 2:i10 ( F270 ) = i43, 3: ARIASG
         VW(#COUNTER,$FLAG[270],10,$COUNT_I[43])
      ;ENDFOLD
      ;FOLD i1 ( EIN ) = 0 ;%{SE}%MKUKATPVW %CVW_SPS %VARIASG %P 2:i1 ( EIN ) = 0, 3: ARIASG
         VW(#COUNTER,TRUE,1,0)
      ;ENDFOLD
      ;FOLD -- Ueberwachungszeit EZ1/SP1/KE1 SZ2 schliessen -- ;%{SE}%MKUKATPVW %CVW_COM %VCOMMENT %P 2:-- Ueberwachungszeit EZ1/SP1/KE1 SZ2 schliessen --, 3: VW_COMMENT
      ;ENDFOLD
      ;FOLD T9 ( EIN ) = -40[1/10Sek] ;%{SE}%MKUKATPVW %CVW_SPS %VTASG %P 2:T9 ( EIN ) = -40[1/10Sek], 3: TASG
         VW(#SET_TIME,TRUE,9,0,-40)
      ;ENDFOLD
      ;FOLD -- Ueberwachungszeit KF1 -- ;%{SE}%MKUKATPVW %CVW_COM %VCOMMENT %P 2:-- Ueberwachungszeit KF1 --, 3: VW_COMMENT
      ;ENDFOLD
      ;FOLD T7 ( EIN ) = -40[1/10Sek] ;%{SE}%MKUKATPVW %CVW_SPS %VTASG %P 2:T7 ( EIN ) = -40[1/10Sek], 3: TASG
         VW(#SET_TIME,TRUE,7,0,-40)
      ;ENDFOLD
      ;FOLD Schritt 21 = A4039  ;%{SE}%MKUKATPVW %CVW_SPS %VST_CON %P 2:Schritt 21 = A4039 , 3: ST_CON
         IF $OUT[4039] THEN
            PREVSTEP = $APP_INT[5]
            $APP_INT[5] = 21
         ENDIF
      ;ENDFOLD
   ;ENDFOLD
   ;FOLD SCHRITT 21 -- ROB EZ1/SP1/KE1 SZ2 -- ;%{P}%MKUKATPVW,%CSTEP,%VST_NR,%P 1:SCHRITT, 2:21, 3: ROB EZ1/SP1/KE1 SZ2
      ;FOLD ;%{H}
         Case 21
      ;ENDFOLD
      ;FOLD F270 = AUS ;%{SE}%MKUKATPVW %CVW_SPS %VBOASG %P 2:F270 = AUS, 3: BOASG
         $FLAG[270] = FALSE
      ;ENDFOLD
      ;FOLD -- KF1/KW1 Ausblasen -- ;%{SE}%MKUKATPVW %CVW_COM %VCOMMENT %P 2:-- KF1/KW1 Ausblasen --, 3: VW_COMMENT
      ;ENDFOLD
      ;FOLD A835 = (F330 + F331 + !F330 & !F331 & !F332) & !F289 & !F72 & !F73 ;%{SE}%MKUKATPVW %CVW_SPS %VBOASG %P 2:A835 = (F330 + F331 + !F330 & !F331 & !F332) & !F289 & !F72 & !F73, 3: BOASG
         $OUT[835] = ($FLAG[330] OR $FLAG[331] OR NOT $FLAG[330] AND NOT $FLAG[331] AND NOT $FLAG[332]) AND NOT $FLAG[289] AND NOT $FLAG[72] AND NOT $FLAG[73]
      ;ENDFOLD
      ;FOLD A859 = (F330 + F331 + !F330 & !F331 & !F332) & F289 & !F72 & !F73 ;%{SE}%MKUKATPVW %CVW_SPS %VBOASG %P 2:A859 = (F330 + F331 + !F330 & !F331 & !F332) & F289 & !F72 & !F73, 3: BOASG
         $OUT[859] = ($FLAG[330] OR $FLAG[331] OR NOT $FLAG[330] AND NOT $FLAG[331] AND NOT $FLAG[332]) AND $FLAG[289] AND NOT $FLAG[72] AND NOT $FLAG[73]
      ;ENDFOLD
      ;FOLD -- KF2/KW2 Ausblasen -- ;%{SE}%MKUKATPVW %CVW_COM %VCOMMENT %P 2:-- KF2/KW2 Ausblasen --, 3: VW_COMMENT
      ;ENDFOLD
      ;FOLD A995 = (F330 + F331 + !F330 & !F331 & !F332) & !F803 & F72 ;%{SE}%MKUKATPVW %CVW_SPS %VBOASG %P 2:A995 = (F330 + F331 + !F330 & !F331 & !F332) & !F803 & F72, 3: BOASG
         $OUT[995] = ($FLAG[330] OR $FLAG[331] OR NOT $FLAG[330] AND NOT $FLAG[331] AND NOT $FLAG[332]) AND NOT $FLAG[803] AND $FLAG[72]
      ;ENDFOLD
      ;FOLD A1019 = (F330 + F331 + !F330 & !F331 & !F332) & F803 & F72 ;%{SE}%MKUKATPVW %CVW_SPS %VBOASG %P 2:A1019 = (F330 + F331 + !F330 & !F331 & !F332) & F803 & F72, 3: BOASG
         $OUT[1019] = ($FLAG[330] OR $FLAG[331] OR NOT $FLAG[330] AND NOT $FLAG[331] AND NOT $FLAG[332]) AND $FLAG[803] AND $FLAG[72]
      ;ENDFOLD
      ;FOLD -- KF3/KW3 Ausblasen ein -- ;%{SE}%MKUKATPVW %CVW_COM %VCOMMENT %P 2:-- KF3/KW3 Ausblasen ein --, 3: VW_COMMENT
      ;ENDFOLD
      ;FOLD A1155 = (F330 + F331 + !F330 & !F331 & !F332) & !F804 & F73 ;%{SE}%MKUKATPVW %CVW_SPS %VBOASG %P 2:A1155 = (F330 + F331 + !F330 & !F331 & !F332) & !F804 & F73, 3: BOASG
         $OUT[1155] = ($FLAG[330] OR $FLAG[331] OR NOT $FLAG[330] AND NOT $FLAG[331] AND NOT $FLAG[332]) AND NOT $FLAG[804] AND $FLAG[73]
      ;ENDFOLD
      ;FOLD A1179 = (F330 + F331 + !F330 & !F331 & !F332) & F804 & F73 ;%{SE}%MKUKATPVW %CVW_SPS %VBOASG %P 2:A1179 = (F330 + F331 + !F330 & !F331 & !F332) & F804 & F73, 3: BOASG
         $OUT[1179] = ($FLAG[330] OR $FLAG[331] OR NOT $FLAG[330] AND NOT $FLAG[331] AND NOT $FLAG[332]) AND $FLAG[804] AND $FLAG[73]
      ;ENDFOLD
      ;FOLD -- EZ1/SP1 SZ1 schliessen -- ;%{SE}%MKUKATPVW %CVW_COM %VCOMMENT %P 2:-- EZ1/SP1 SZ1 schliessen --, 3: VW_COMMENT
      ;ENDFOLD
      ;FOLD A717 = AUS ;%{SE}%MKUKATPVW %CVW_SPS %VBOASG %P 2:A717 = AUS, 3: BOASG
         $OUT[717] = FALSE
      ;ENDFOLD
      ;FOLD A718 = EIN ;%{SE}%MKUKATPVW %CVW_SPS %VBOASG %P 2:A718 = EIN, 3: BOASG
         $OUT[718] = TRUE
      ;ENDFOLD
      ;FOLD Schritt 22 = (!E717 & E718 + T9) & A4039  ;%{SE}%MKUKATPVW %CVW_SPS %VST_CON %P 2:Schritt 22 = (!E717 & E718 + T9) & A4039 , 3: ST_CON
         IF (NOT $IN[717] AND $IN[718] OR $TIMER_FLAG[9]) AND $OUT[4039] THEN
            PREVSTEP = $APP_INT[5]
            $APP_INT[5] = 22
         ENDIF
      ;ENDFOLD
   ;ENDFOLD
   ;FOLD SCHRITT 22 -- ROB EZ1/SP1/KE1 SZ2 -- ;%{P}%MKUKATPVW,%CSTEP,%VST_NR,%P 1:SCHRITT, 2:22, 3: ROB EZ1/SP1/KE1 SZ2
      ;FOLD ;%{H}
         Case 22
      ;ENDFOLD
      ;FOLD T9 ( EIN ) = STOP ;%{SE}%MKUKATPVW %CVW_SPS %VTSTOP %P 2:T9 ( EIN ) = STOP, 3: TSTOP
         VW(#SET_TIME,TRUE,9,1,0)
      ;ENDFOLD
      ;FOLD -- RSK Fehlerausgabe Kraftaufbau -- ;%{SE}%MKUKATPVW %CVW_COM %VCOMMENT %P 2:-- RSK Fehlerausgabe Kraftaufbau --, 3: VW_COMMENT
      ;ENDFOLD
      ;FOLD F325 = T9 ;%{SE}%MKUKATPVW %CVW_SPS %VBOASG %P 2:F325 = T9, 3: BOASG
         $FLAG[325] = $TIMER_FLAG[9]
      ;ENDFOLD
      ;FOLD -- KF1/KW1 abschalten bei Fehler -- ;%{SE}%MKUKATPVW %CVW_COM %VCOMMENT %P 2:-- KF1/KW1 abschalten bei Fehler --, 3: VW_COMMENT
      ;ENDFOLD
      ;FOLD A834 = A834 & !T7 & !T9 & !F289 & !F72 & !F73 ;%{SE}%MKUKATPVW %CVW_SPS %VBOASG %P 2:A834 = A834 & !T7 & !T9 & !F289 & !F72 & !F73, 3: BOASG
         $OUT[834] = $OUT[834] AND NOT $TIMER_FLAG[7] AND NOT $TIMER_FLAG[9] AND NOT $FLAG[289] AND NOT $FLAG[72] AND NOT $FLAG[73]
      ;ENDFOLD
      ;FOLD A858 = A858 & !T7 & !T9 & F289 & !F72 & !F73 ;%{SE}%MKUKATPVW %CVW_SPS %VBOASG %P 2:A858 = A858 & !T7 & !T9 & F289 & !F72 & !F73, 3: BOASG
         $OUT[858] = $OUT[858] AND NOT $TIMER_FLAG[7] AND NOT $TIMER_FLAG[9] AND $FLAG[289] AND NOT $FLAG[72] AND NOT $FLAG[73]
      ;ENDFOLD
      ;FOLD -- KF2/KW2 abschalten bei Fehler -- ;%{SE}%MKUKATPVW %CVW_COM %VCOMMENT %P 2:-- KF2/KW2 abschalten bei Fehler --, 3: VW_COMMENT
      ;ENDFOLD
      ;FOLD A994 = A994 & !T7 & !T9 & !F803 & F72 ;%{SE}%MKUKATPVW %CVW_SPS %VBOASG %P 2:A994 = A994 & !T7 & !T9 & !F803 & F72, 3: BOASG
         $OUT[994] = $OUT[994] AND NOT $TIMER_FLAG[7] AND NOT $TIMER_FLAG[9] AND NOT $FLAG[803] AND $FLAG[72]
      ;ENDFOLD
      ;FOLD A1018 = A1018 & !T7 & !T9 & F803 & F72 ;%{SE}%MKUKATPVW %CVW_SPS %VBOASG %P 2:A1018 = A1018 & !T7 & !T9 & F803 & F72, 3: BOASG
         $OUT[1018] = $OUT[1018] AND NOT $TIMER_FLAG[7] AND NOT $TIMER_FLAG[9] AND $FLAG[803] AND $FLAG[72]
      ;ENDFOLD
      ;FOLD -- KF3/KW3 abschalten bei Fehler -- ;%{SE}%MKUKATPVW %CVW_COM %VCOMMENT %P 2:-- KF3/KW3 abschalten bei Fehler --, 3: VW_COMMENT
      ;ENDFOLD
      ;FOLD A1154 = A1154 & !T7 & !T9 & !F804 & F73 ;%{SE}%MKUKATPVW %CVW_SPS %VBOASG %P 2:A1154 = A1154 & !T7 & !T9 & !F804 & F73, 3: BOASG
         $OUT[1154] = $OUT[1154] AND NOT $TIMER_FLAG[7] AND NOT $TIMER_FLAG[9] AND NOT $FLAG[804] AND $FLAG[73]
      ;ENDFOLD
      ;FOLD A1178 = A1178 & !T7 & !T9 & F804 & F73 ;%{SE}%MKUKATPVW %CVW_SPS %VBOASG %P 2:A1178 = A1178 & !T7 & !T9 & F804 & F73, 3: BOASG
         $OUT[1178] = $OUT[1178] AND NOT $TIMER_FLAG[7] AND NOT $TIMER_FLAG[9] AND $FLAG[804] AND $FLAG[73]
      ;ENDFOLD
      ;FOLD -- KF1/KW1 Ausblasen -- ;%{SE}%MKUKATPVW %CVW_COM %VCOMMENT %P 2:-- KF1/KW1 Ausblasen --, 3: VW_COMMENT
      ;ENDFOLD
      ;FOLD A835 = (F330 + F331 + !F330 & !F331 & !F332) & !T9 & !F289 & !F72 & !F73 ;%{SE}%MKUKATPVW %CVW_SPS %VBOASG %P 2:A835 = (F330 + F331 + !F330 & !F331 & !F332) & !T9 & !F289 & !F72 & !F73, 3: BOASG
         $OUT[835] = ($FLAG[330] OR $FLAG[331] OR NOT $FLAG[330] AND NOT $FLAG[331] AND NOT $FLAG[332]) AND NOT $TIMER_FLAG[9] AND NOT $FLAG[289] AND NOT $FLAG[72] AND NOT $FLAG[73]
      ;ENDFOLD
      ;FOLD A859 = (F330 + F331 + !F330 & !F331 & !F332) & !T9 & F289 & !F72 & !F73 ;%{SE}%MKUKATPVW %CVW_SPS %VBOASG %P 2:A859 = (F330 + F331 + !F330 & !F331 & !F332) & !T9 & F289 & !F72 & !F73, 3: BOASG
         $OUT[859] = ($FLAG[330] OR $FLAG[331] OR NOT $FLAG[330] AND NOT $FLAG[331] AND NOT $FLAG[332]) AND NOT $TIMER_FLAG[9] AND $FLAG[289] AND NOT $FLAG[72] AND NOT $FLAG[73]
      ;ENDFOLD
      ;FOLD -- KF2/KW2 Ausblasen -- ;%{SE}%MKUKATPVW %CVW_COM %VCOMMENT %P 2:-- KF2/KW2 Ausblasen --, 3: VW_COMMENT
      ;ENDFOLD
      ;FOLD A995 = (F330 + F331 + !F330 & !F331 & !F332) & !T9 & !F803 & F72 ;%{SE}%MKUKATPVW %CVW_SPS %VBOASG %P 2:A995 = (F330 + F331 + !F330 & !F331 & !F332) & !T9 & !F803 & F72, 3: BOASG
         $OUT[995] = ($FLAG[330] OR $FLAG[331] OR NOT $FLAG[330] AND NOT $FLAG[331] AND NOT $FLAG[332]) AND NOT $TIMER_FLAG[9] AND NOT $FLAG[803] AND $FLAG[72]
      ;ENDFOLD
      ;FOLD A1019 = (F330 + F331 + !F330 & !F331 & !F332) & !T9 & F803 & F72 ;%{SE}%MKUKATPVW %CVW_SPS %VBOASG %P 2:A1019 = (F330 + F331 + !F330 & !F331 & !F332) & !T9 & F803 & F72, 3: BOASG
         $OUT[1019] = ($FLAG[330] OR $FLAG[331] OR NOT $FLAG[330] AND NOT $FLAG[331] AND NOT $FLAG[332]) AND NOT $TIMER_FLAG[9] AND $FLAG[803] AND $FLAG[72]
      ;ENDFOLD
      ;FOLD -- KF3/KW3 Ausblasen -- ;%{SE}%MKUKATPVW %CVW_COM %VCOMMENT %P 2:-- KF3/KW3 Ausblasen --, 3: VW_COMMENT
      ;ENDFOLD
      ;FOLD A1155 = (F330 + F331 + !F330 & !F331 & !F332) & !F804 & F73 ;%{SE}%MKUKATPVW %CVW_SPS %VBOASG %P 2:A1155 = (F330 + F331 + !F330 & !F331 & !F332) & !F804 & F73, 3: BOASG
         $OUT[1155] = ($FLAG[330] OR $FLAG[331] OR NOT $FLAG[330] AND NOT $FLAG[331] AND NOT $FLAG[332]) AND NOT $FLAG[804] AND $FLAG[73]
      ;ENDFOLD
      ;FOLD A1179 = (F330 + F331 + !F330 & !F331 & !F332) & F804 & F73 ;%{SE}%MKUKATPVW %CVW_SPS %VBOASG %P 2:A1179 = (F330 + F331 + !F330 & !F331 & !F332) & F804 & F73, 3: BOASG
         $OUT[1179] = ($FLAG[330] OR $FLAG[331] OR NOT $FLAG[330] AND NOT $FLAG[331] AND NOT $FLAG[332]) AND $FLAG[804] AND $FLAG[73]
      ;ENDFOLD
      ;FOLD -- Warte Fraesen fertig oder Timeout -- ;%{SE}%MKUKATPVW %CVW_COM %VCOMMENT %P 2:-- Warte Fraesen fertig oder Timeout --, 3: VW_COMMENT
      ;ENDFOLD
      ;FOLD Schritt 23 = (F79 & F104 + F78 & F100 & !F287 + F78 & F102 & F287 + T7 + T9) & A4039  ;%{SE}%MKUKATPVW %CVW_SPS %VST_CON %P 2:Schritt 23 = (F79 & F104 + F78 & F100 & !F287 + F78 & F102 & F287 + T7 + T9) & A4039 , 3: ST_CON
         IF ($FLAG[79] AND $FLAG[104] OR $FLAG[78] AND $FLAG[100] AND NOT $FLAG[287] OR $FLAG[78] AND $FLAG[102] AND $FLAG[287] OR $TIMER_FLAG[7] OR $TIMER_FLAG[9]) AND $OUT[4039] THEN
            PREVSTEP = $APP_INT[5]
            $APP_INT[5] = 23
         ENDIF
      ;ENDFOLD
   ;ENDFOLD
   ;FOLD SCHRITT 23 -- ROB EZ1/SP1/KE1 SZ2 -- ;%{P}%MKUKATPVW,%CSTEP,%VST_NR,%P 1:SCHRITT, 2:23, 3: ROB EZ1/SP1/KE1 SZ2
      ;FOLD ;%{H}
         Case 23
      ;ENDFOLD
      ;FOLD t7 ( EIN ) = STOP ;%{SE}%MKUKATPVW %CVW_SPS %VTSTOP %P 2:t7 ( EIN ) = STOP, 3: TSTOP
         VW(#SET_TIME,TRUE,7,1,0)
      ;ENDFOLD
      ;FOLD -- Hilfsflag SK Programmwechsel -- ;%{SE}%MKUKATPVW %CVW_COM %VCOMMENT %P 2:-- Hilfsflag SK Programmwechsel --, 3: VW_COMMENT
      ;ENDFOLD
      ;FOLD F334 = AUS ;%{SE}%MKUKATPVW %CVW_SPS %VBOASG %P 2:F334 = AUS, 3: BOASG
         $FLAG[334] = FALSE
      ;ENDFOLD
      ;FOLD -- EZ1/SP1 SZ2 oeffnen -- ;%{SE}%MKUKATPVW %CVW_COM %VCOMMENT %P 2:-- EZ1/SP1 SZ2 oeffnen --, 3: VW_COMMENT
      ;ENDFOLD
      ;FOLD A719 = AUS ;%{SE}%MKUKATPVW %CVW_SPS %VBOASG %P 2:A719 = AUS, 3: BOASG
         $OUT[719] = FALSE
      ;ENDFOLD
      ;FOLD A718 = AUS ;%{SE}%MKUKATPVW %CVW_SPS %VBOASG %P 2:A718 = AUS, 3: BOASG
         $OUT[718] = FALSE
      ;ENDFOLD
      ;FOLD A717 = EIN ;%{SE}%MKUKATPVW %CVW_SPS %VBOASG %P 2:A717 = EIN, 3: BOASG
         $OUT[717] = TRUE
      ;ENDFOLD
      ;FOLD -- KF1/KW1 Ausblasen -- ;%{SE}%MKUKATPVW %CVW_COM %VCOMMENT %P 2:-- KF1/KW1 Ausblasen --, 3: VW_COMMENT
      ;ENDFOLD
      ;FOLD A835 = (F330 + F331 + F332 + !F330 & !F331 & !F332) & !F289 & !F72 & !F73 ;%{SE}%MKUKATPVW %CVW_SPS %VBOASG %P 2:A835 = (F330 + F331 + F332 + !F330 & !F331 & !F332) & !F289 & !F72 & !F73, 3: BOASG
         $OUT[835] = ($FLAG[330] OR $FLAG[331] OR $FLAG[332] OR NOT $FLAG[330] AND NOT $FLAG[331] AND NOT $FLAG[332]) AND NOT $FLAG[289] AND NOT $FLAG[72] AND NOT $FLAG[73]
      ;ENDFOLD
      ;FOLD A859 = (F330 + F331 + F332 + !F330 & !F331 & !F332) & F289 & !F72 & !F73 ;%{SE}%MKUKATPVW %CVW_SPS %VBOASG %P 2:A859 = (F330 + F331 + F332 + !F330 & !F331 & !F332) & F289 & !F72 & !F73, 3: BOASG
         $OUT[859] = ($FLAG[330] OR $FLAG[331] OR $FLAG[332] OR NOT $FLAG[330] AND NOT $FLAG[331] AND NOT $FLAG[332]) AND $FLAG[289] AND NOT $FLAG[72] AND NOT $FLAG[73]
      ;ENDFOLD
      ;FOLD -- KF2/KW2 Ausblasen -- ;%{SE}%MKUKATPVW %CVW_COM %VCOMMENT %P 2:-- KF2/KW2 Ausblasen --, 3: VW_COMMENT
      ;ENDFOLD
      ;FOLD A995 = (F330 + F331 + F332 + !F330 & !F331 & !F332) & !F803 & F72 ;%{SE}%MKUKATPVW %CVW_SPS %VBOASG %P 2:A995 = (F330 + F331 + F332 + !F330 & !F331 & !F332) & !F803 & F72, 3: BOASG
         $OUT[995] = ($FLAG[330] OR $FLAG[331] OR $FLAG[332] OR NOT $FLAG[330] AND NOT $FLAG[331] AND NOT $FLAG[332]) AND NOT $FLAG[803] AND $FLAG[72]
      ;ENDFOLD
      ;FOLD A1019 = (F330 + F331 + F332 + !F330 & !F331 & !F332) & F803 & F72 ;%{SE}%MKUKATPVW %CVW_SPS %VBOASG %P 2:A1019 = (F330 + F331 + F332 + !F330 & !F331 & !F332) & F803 & F72, 3: BOASG
         $OUT[1019] = ($FLAG[330] OR $FLAG[331] OR $FLAG[332] OR NOT $FLAG[330] AND NOT $FLAG[331] AND NOT $FLAG[332]) AND $FLAG[803] AND $FLAG[72]
      ;ENDFOLD
      ;FOLD -- KF3/KW3 Ausblasen ein -- ;%{SE}%MKUKATPVW %CVW_COM %VCOMMENT %P 2:-- KF3/KW3 Ausblasen ein --, 3: VW_COMMENT
      ;ENDFOLD
      ;FOLD A1155 = (F330 + F331 + F332 & !F330 & !F331 & !F332) & !F804 & F73 ;%{SE}%MKUKATPVW %CVW_SPS %VBOASG %P 2:A1155 = (F330 + F331 + F332 & !F330 & !F331 & !F332) & !F804 & F73, 3: BOASG
         $OUT[1155] = ($FLAG[330] OR $FLAG[331] OR $FLAG[332] AND NOT $FLAG[330] AND NOT $FLAG[331] AND NOT $FLAG[332]) AND NOT $FLAG[804] AND $FLAG[73]
      ;ENDFOLD
      ;FOLD A1179 = (F330 + F331 + F332 & !F330 & !F331 & !F332) & F804 & F73 ;%{SE}%MKUKATPVW %CVW_SPS %VBOASG %P 2:A1179 = (F330 + F331 + F332 & !F330 & !F331 & !F332) & F804 & F73, 3: BOASG
         $OUT[1179] = ($FLAG[330] OR $FLAG[331] OR $FLAG[332] AND NOT $FLAG[330] AND NOT $FLAG[331] AND NOT $FLAG[332]) AND $FLAG[804] AND $FLAG[73]
      ;ENDFOLD
      ;FOLD -- RSK Sammelstoerung -- ;%{SE}%MKUKATPVW %CVW_COM %VCOMMENT %P 2:-- RSK Sammelstoerung --, 3: VW_COMMENT
      ;ENDFOLD
      ;FOLD F329 = T7 + T9 ;%{SE}%MKUKATPVW %CVW_SPS %VBOASG %P 2:F329 = T7 + T9, 3: BOASG
         $FLAG[329] = $TIMER_FLAG[7] OR $TIMER_FLAG[9]
      ;ENDFOLD
      ;FOLD -- Hilfsflag Startfraesen -- ;%{SE}%MKUKATPVW %CVW_COM %VCOMMENT %P 2:-- Hilfsflag Startfraesen --, 3: VW_COMMENT
      ;ENDFOLD
      ;FOLD F102 = (F102 & F78 + F104 & F79) & F287 ;%{SE}%MKUKATPVW %CVW_SPS %VBOASG %P 2:F102 = (F102 & F78 + F104 & F79) & F287, 3: BOASG
         $FLAG[102] = ($FLAG[102] AND $FLAG[78] OR $FLAG[104] AND $FLAG[79]) AND $FLAG[287]
      ;ENDFOLD
      ;FOLD F104 = !F130 & F104 + F130 & F287 & F104 ;%{SE}%MKUKATPVW %CVW_SPS %VBOASG %P 2:F104 = !F130 & F104 + F130 & F287 & F104, 3: BOASG
         $FLAG[104] = NOT $FLAG[130] AND $FLAG[104] OR $FLAG[130] AND $FLAG[287] AND $FLAG[104]
      ;ENDFOLD
      ;FOLD F287 = F78 + F79 & F130 ;%{SE}%MKUKATPVW %CVW_SPS %VBOASG %P 2:F287 = F78 + F79 & F130, 3: BOASG
         $FLAG[287] = $FLAG[78] OR $FLAG[79] AND $FLAG[130]
      ;ENDFOLD
      ;FOLD -- Neues Fraesprogramm und Zaehler ruecksetzen -- ;%{SE}%MKUKATPVW %CVW_COM %VCOMMENT %P 2:-- Neues Fraesprogramm und Zaehler ruecksetzen --, 3: VW_COMMENT
      ;ENDFOLD
      ;FOLD F270 = F102 & F732 ;%{SE}%MKUKATPVW %CVW_SPS %VBOASG %P 2:F270 = F102 & F732, 3: BOASG
         $FLAG[270] = $FLAG[102] AND $FLAG[732]
      ;ENDFOLD
      ;FOLD bin3 ( F732 ) = 37 ;%{SE}%MKUKATPVW %CVW_SPS %VARIASG %P 2:bin3 ( F732 ) = 37, 3: ARIASG
         VW(#BINOUT,$FLAG[732],3,37)
      ;ENDFOLD
      ;FOLD i10 ( F270 ) = i45 ;%{SE}%MKUKATPVW %CVW_SPS %VARIASG %P 2:i10 ( F270 ) = i45, 3: ARIASG
         VW(#COUNTER,$FLAG[270],10,$COUNT_I[45])
      ;ENDFOLD
      ;FOLD -- Wiederholung beim Startfraesen -- ;%{SE}%MKUKATPVW %CVW_COM %VCOMMENT %P 2:-- Wiederholung beim Startfraesen --, 3: VW_COMMENT
      ;ENDFOLD
      ;FOLD Schritt 20 = E717 & !E718 & (F78 & !F102 + F79 & F130 & !F102) & !F329 & A4039  ;%{SE}%MKUKATPVW %CVW_SPS %VST_CON %P 2:Schritt 20 = E717 & !E718 & (F78 & !F102 + F79 & F130 & !F102) & !F329 & A4039 , 3: ST_CON
         IF $IN[717] AND NOT $IN[718] AND ($FLAG[78] AND NOT $FLAG[102] OR $FLAG[79] AND $FLAG[130] AND NOT $FLAG[102]) AND NOT $FLAG[329] AND $OUT[4039] THEN
            PREVSTEP = $APP_INT[5]
            $APP_INT[5] = 20
         ENDIF
      ;ENDFOLD
      ;FOLD -- Weiter wenn Fraesen fertig -- ;%{SE}%MKUKATPVW %CVW_COM %VCOMMENT %P 2:-- Weiter wenn Fraesen fertig --, 3: VW_COMMENT
      ;ENDFOLD
      ;FOLD Schritt 24 = E717 & !E718 & (F79 & F104 & (!F130 + F102) + F78 & F102 + F329) & A4039  ;%{SE}%MKUKATPVW %CVW_SPS %VST_CON %P 2:Schritt 24 = E717 & !E718 & (F79 & F104 & (!F130 + F102) + F78 & F102 + F329) & A4039 , 3: ST_CON
         IF $IN[717] AND NOT $IN[718] AND ($FLAG[79] AND $FLAG[104] AND (NOT $FLAG[130] OR $FLAG[102]) OR $FLAG[78] AND $FLAG[102] OR $FLAG[329]) AND $OUT[4039] THEN
            PREVSTEP = $APP_INT[5]
            $APP_INT[5] = 24
         ENDIF
      ;ENDFOLD
      ;FOLD -- Weiter bei Fehler -- ;%{SE}%MKUKATPVW %CVW_COM %VCOMMENT %P 2:-- Weiter bei Fehler --, 3: VW_COMMENT
      ;ENDFOLD
      ;FOLD Schritt 26 = F325 & (E26 + E27) & A4039  ;%{SE}%MKUKATPVW %CVW_SPS %VST_CON %P 2:Schritt 26 = F325 & (E26 + E27) & A4039 , 3: ST_CON
         IF $FLAG[325] AND ($IN[26] OR $IN[27]) AND $OUT[4039] THEN
            PREVSTEP = $APP_INT[5]
            $APP_INT[5] = 26
         ENDIF
      ;ENDFOLD
   ;ENDFOLD
   ;FOLD SCHRITT 24 -- ROB EZ1/SP1/KE1 SZ2 -- ;%{P}%MKUKATPVW,%CSTEP,%VST_NR,%P 1:SCHRITT, 2:24, 3: ROB EZ1/SP1/KE1 SZ2
      ;FOLD ;%{H}
         Case 24
      ;ENDFOLD
      ;FOLD F270 = AUS ;%{SE}%MKUKATPVW %CVW_SPS %VBOASG %P 2:F270 = AUS, 3: BOASG
         $FLAG[270] = FALSE
      ;ENDFOLD
      ;FOLD A717 = AUS ;%{SE}%MKUKATPVW %CVW_SPS %VBOASG %P 2:A717 = AUS, 3: BOASG
         $OUT[717] = FALSE
      ;ENDFOLD
      ;FOLD -- KF1/KW1 abschalten -- ;%{SE}%MKUKATPVW %CVW_COM %VCOMMENT %P 2:-- KF1/KW1 abschalten --, 3: VW_COMMENT
      ;ENDFOLD
      ;FOLD A834 = AUS ;%{SE}%MKUKATPVW %CVW_SPS %VBOASG %P 2:A834 = AUS, 3: BOASG
         $OUT[834] = FALSE
      ;ENDFOLD
      ;FOLD A858 = AUS ;%{SE}%MKUKATPVW %CVW_SPS %VBOASG %P 2:A858 = AUS, 3: BOASG
         $OUT[858] = FALSE
      ;ENDFOLD
      ;FOLD -- KF2/KW2 abschalten -- ;%{SE}%MKUKATPVW %CVW_COM %VCOMMENT %P 2:-- KF2/KW2 abschalten --, 3: VW_COMMENT
      ;ENDFOLD
      ;FOLD A994 = AUS ;%{SE}%MKUKATPVW %CVW_SPS %VBOASG %P 2:A994 = AUS, 3: BOASG
         $OUT[994] = FALSE
      ;ENDFOLD
      ;FOLD A1018 = AUS ;%{SE}%MKUKATPVW %CVW_SPS %VBOASG %P 2:A1018 = AUS, 3: BOASG
         $OUT[1018] = FALSE
      ;ENDFOLD
      ;FOLD -- KF3/KW3 abschalten -- ;%{SE}%MKUKATPVW %CVW_COM %VCOMMENT %P 2:-- KF3/KW3 abschalten --, 3: VW_COMMENT
      ;ENDFOLD
      ;FOLD A1154 = AUS ;%{SE}%MKUKATPVW %CVW_SPS %VBOASG %P 2:A1154 = AUS, 3: BOASG
         $OUT[1154] = FALSE
      ;ENDFOLD
      ;FOLD A1178 = AUS ;%{SE}%MKUKATPVW %CVW_SPS %VBOASG %P 2:A1178 = AUS, 3: BOASG
         $OUT[1178] = FALSE
      ;ENDFOLD
      ;FOLD bin3 ( !F329 ) = 2 ;%{SE}%MKUKATPVW %CVW_SPS %VARIASG %P 2:bin3 ( !F329 ) = 2, 3: ARIASG
         VW(#BINOUT,NOT $FLAG[329],3,2)
      ;ENDFOLD
      ;FOLD -- Wartezeit Programmwechsel SK -- ;%{SE}%MKUKATPVW %CVW_COM %VCOMMENT %P 2:-- Wartezeit Programmwechsel SK --, 3: VW_COMMENT
      ;ENDFOLD
      ;FOLD T8 ( !F334 ) = -2[1/10Sek] ;%{SE}%MKUKATPVW %CVW_SPS %VTASG %P 2:T8 ( !F334 ) = -2[1/10Sek], 3: TASG
         VW(#SET_TIME,NOT $FLAG[334],8,0,-2)
      ;ENDFOLD
      ;FOLD -- Hilfsflag SK Programmwechsel -- ;%{SE}%MKUKATPVW %CVW_COM %VCOMMENT %P 2:-- Hilfsflag SK Programmwechsel --, 3: VW_COMMENT
      ;ENDFOLD
      ;FOLD F334 = EIN ;%{SE}%MKUKATPVW %CVW_SPS %VBOASG %P 2:F334 = EIN, 3: BOASG
         $FLAG[334] = TRUE
      ;ENDFOLD
      ;FOLD Schritt 25 = T8 & A4039  ;%{SE}%MKUKATPVW %CVW_SPS %VST_CON %P 2:Schritt 25 = T8 & A4039 , 3: ST_CON
         IF $TIMER_FLAG[8] AND $OUT[4039] THEN
            PREVSTEP = $APP_INT[5]
            $APP_INT[5] = 25
         ENDIF
      ;ENDFOLD
   ;ENDFOLD
   ;FOLD SCHRITT 25 -- ROB EZ1/SP1 SZ2 -- ;%{P}%MKUKATPVW,%CSTEP,%VST_NR,%P 1:SCHRITT, 2:25, 3: ROB EZ1/SP1 SZ2
      ;FOLD ;%{H}
         Case 25
      ;ENDFOLD
      ;FOLD -- Hilfsflag SK Programmwechsel -- ;%{SE}%MKUKATPVW %CVW_COM %VCOMMENT %P 2:-- Hilfsflag SK Programmwechsel --, 3: VW_COMMENT
      ;ENDFOLD
      ;FOLD F334 = AUS ;%{SE}%MKUKATPVW %CVW_SPS %VBOASG %P 2:F334 = AUS, 3: BOASG
         $FLAG[334] = FALSE
      ;ENDFOLD
      ;FOLD -- Quitt. Fraesen SK1 -- ;%{SE}%MKUKATPVW %CVW_COM %VCOMMENT %P 2:-- Quitt. Fraesen SK1 --, 3: VW_COMMENT
      ;ENDFOLD
      ;FOLD A786 = (!F329 & !F322 & !F830) + (F830 & A786) ;%{SE}%MKUKATPVW %CVW_SPS %VBOASG %P 2:A786 = (!F329 & !F322 & !F830) + (F830 & A786), 3: BOASG
         $OUT[786] = (NOT $FLAG[329] AND NOT $FLAG[322] AND NOT $FLAG[830]) OR ($FLAG[830] AND $OUT[786])
      ;ENDFOLD
      ;FOLD A722 = (!F329 & !F322 & F830) + (!F830 & A722) ;%{SE}%MKUKATPVW %CVW_SPS %VBOASG %P 2:A722 = (!F329 & !F322 & F830) + (!F830 & A722), 3: BOASG
         $OUT[722] = (NOT $FLAG[329] AND NOT $FLAG[322] AND $FLAG[830]) OR (NOT $FLAG[830] AND $OUT[722])
      ;ENDFOLD
      ;FOLD Schritt 26 = (!F830 & !E786 & E787 & !E788 + F830 & !E722 & E724 & !E723 + F329) & A4039  ;%{SE}%MKUKATPVW %CVW_SPS %VST_CON %P 2:Schritt 26 = (!F830 & !E786 & E787 & !E788 + F830 & !E722 & E724 & !E723 + F329) & A4039 , 3: ST_CON
         IF (NOT $FLAG[830] AND NOT $IN[786] AND $IN[787] AND NOT $IN[788] OR $FLAG[830] AND NOT $IN[722] AND $IN[724] AND NOT $IN[723] OR $FLAG[329]) AND $OUT[4039] THEN
            PREVSTEP = $APP_INT[5]
            $APP_INT[5] = 26
         ENDIF
      ;ENDFOLD
   ;ENDFOLD
   ;FOLD SCHRITT 26 -- ROB EZ1/SP1/KE1 SZ2 # Ende -- ;%{P}%MKUKATPVW,%CSTEP,%VST_NR,%P 1:SCHRITT, 2:26, 3: ROB EZ1/SP1/KE1 SZ2 # Ende
      ;FOLD ;%{H}
         Case 26
      ;ENDFOLD
      ;FOLD F270 = AUS ;%{SE}%MKUKATPVW %CVW_SPS %VBOASG %P 2:F270 = AUS, 3: BOASG
         $FLAG[270] = FALSE
      ;ENDFOLD
      ;FOLD -- KF1/KW1 Ausblasen -- ;%{SE}%MKUKATPVW %CVW_COM %VCOMMENT %P 2:-- KF1/KW1 Ausblasen --, 3: VW_COMMENT
      ;ENDFOLD
      ;FOLD A835 = (F330 + F331 + F332) & F736 & !F72 & !F73 ;%{SE}%MKUKATPVW %CVW_SPS %VBOASG %P 2:A835 = (F330 + F331 + F332) & F736 & !F72 & !F73, 3: BOASG
         $OUT[835] = ($FLAG[330] OR $FLAG[331] OR $FLAG[332]) AND $FLAG[736] AND NOT $FLAG[72] AND NOT $FLAG[73]
      ;ENDFOLD
      ;FOLD A859 = (F330 + F331 + F332) & F736 & !F72 & !F73 ;%{SE}%MKUKATPVW %CVW_SPS %VBOASG %P 2:A859 = (F330 + F331 + F332) & F736 & !F72 & !F73, 3: BOASG
         $OUT[859] = ($FLAG[330] OR $FLAG[331] OR $FLAG[332]) AND $FLAG[736] AND NOT $FLAG[72] AND NOT $FLAG[73]
      ;ENDFOLD
      ;FOLD -- KF2/KW2 Ausblasen -- ;%{SE}%MKUKATPVW %CVW_COM %VCOMMENT %P 2:-- KF2/KW2 Ausblasen --, 3: VW_COMMENT
      ;ENDFOLD
      ;FOLD A995 = (F330 + F331 + F332) & F736 & F72 ;%{SE}%MKUKATPVW %CVW_SPS %VBOASG %P 2:A995 = (F330 + F331 + F332) & F736 & F72, 3: BOASG
         $OUT[995] = ($FLAG[330] OR $FLAG[331] OR $FLAG[332]) AND $FLAG[736] AND $FLAG[72]
      ;ENDFOLD
      ;FOLD A1019 = (F330 + F331 + F332) & F736 & F72 ;%{SE}%MKUKATPVW %CVW_SPS %VBOASG %P 2:A1019 = (F330 + F331 + F332) & F736 & F72, 3: BOASG
         $OUT[1019] = ($FLAG[330] OR $FLAG[331] OR $FLAG[332]) AND $FLAG[736] AND $FLAG[72]
      ;ENDFOLD
      ;FOLD -- KF3/KW3 Ausblasen -- ;%{SE}%MKUKATPVW %CVW_COM %VCOMMENT %P 2:-- KF3/KW3 Ausblasen --, 3: VW_COMMENT
      ;ENDFOLD
      ;FOLD A1154 = (F330 + F331 + F332) & F736 & F73 ;%{SE}%MKUKATPVW %CVW_SPS %VBOASG %P 2:A1154 = (F330 + F331 + F332) & F736 & F73, 3: BOASG
         $OUT[1154] = ($FLAG[330] OR $FLAG[331] OR $FLAG[332]) AND $FLAG[736] AND $FLAG[73]
      ;ENDFOLD
      ;FOLD A1178 = (F330 + F331 + F332) & F736 & F73 ;%{SE}%MKUKATPVW %CVW_SPS %VBOASG %P 2:A1178 = (F330 + F331 + F332) & F736 & F73, 3: BOASG
         $OUT[1178] = ($FLAG[330] OR $FLAG[331] OR $FLAG[332]) AND $FLAG[736] AND $FLAG[73]
      ;ENDFOLD
      ;FOLD F91 = (!E786 & E787 & !E788 & !F830 + !E722 & E724 & !E723 & F830) & !F322 & !F325 & !F329 ;%{SE}%MKUKATPVW %CVW_SPS %VBOASG %P 2:F91 = (!E786 & E787 & !E788 & !F830 + !E722 & E724 & !E723 & F830) & !F322 & !F325 & !F329, 3: BOASG
         $FLAG[91] = (NOT $IN[786] AND $IN[787] AND NOT $IN[788] AND NOT $FLAG[830] OR NOT $IN[722] AND $IN[724] AND NOT $IN[723] AND $FLAG[830]) AND NOT $FLAG[322] AND NOT $FLAG[325] AND NOT $FLAG[329]
      ;ENDFOLD
      ;FOLD Schritt 15 = (F322 + F325 + F329) & (E26 + E27) & A4039  ;%{SE}%MKUKATPVW %CVW_SPS %VST_CON %P 2:Schritt 15 = (F322 + F325 + F329) & (E26 + E27) & A4039 , 3: ST_CON
         IF ($FLAG[322] OR $FLAG[325] OR $FLAG[329]) AND ($IN[26] OR $IN[27]) AND $OUT[4039] THEN
            PREVSTEP = $APP_INT[5]
            $APP_INT[5] = 15
         ENDIF
      ;ENDFOLD
      ;FOLD Schritt 1 = F91 & !F322 & !F325 & !F329 & A4039  ;%{SE}%MKUKATPVW %CVW_SPS %VST_CON %P 2:Schritt 1 = F91 & !F322 & !F325 & !F329 & A4039 , 3: ST_CON
         IF $FLAG[91] AND NOT $FLAG[322] AND NOT $FLAG[325] AND NOT $FLAG[329] AND $OUT[4039] THEN
            PREVSTEP = $APP_INT[5]
            $APP_INT[5] = 1
         ENDIF
      ;ENDFOLD
   ;ENDFOLD
   ;FOLD SCHRITT 27 -- ROB EZ1/SP1/KE1 SZ3 # Start-- ;%{P}%MKUKATPVW,%CSTEP,%VST_NR,%P 1:SCHRITT, 2:27, 3: ROB EZ1/SP1/KE1 SZ3 # Start
      ;FOLD ;%{H}
         Case 27
      ;ENDFOLD
      ;FOLD -- RSK gestartet -- ;%{SE}%MKUKATPVW %CVW_COM %VCOMMENT %P 2:-- RSK gestartet --, 3: VW_COMMENT
      ;ENDFOLD
      ;FOLD F321 = AUS ;%{SE}%MKUKATPVW %CVW_SPS %VBOASG %P 2:F321 = AUS, 3: BOASG
         $FLAG[321] = FALSE
      ;ENDFOLD
      ;FOLD F322 = AUS ;%{SE}%MKUKATPVW %CVW_SPS %VBOASG %P 2:F322 = AUS, 3: BOASG
         $FLAG[322] = FALSE
      ;ENDFOLD
      ;FOLD F323 = AUS ;%{SE}%MKUKATPVW %CVW_SPS %VBOASG %P 2:F323 = AUS, 3: BOASG
         $FLAG[323] = FALSE
      ;ENDFOLD
      ;FOLD F324 = AUS ;%{SE}%MKUKATPVW %CVW_SPS %VBOASG %P 2:F324 = AUS, 3: BOASG
         $FLAG[324] = FALSE
      ;ENDFOLD
      ;FOLD F325 = AUS ;%{SE}%MKUKATPVW %CVW_SPS %VBOASG %P 2:F325 = AUS, 3: BOASG
         $FLAG[325] = FALSE
      ;ENDFOLD
      ;FOLD F327 = AUS ;%{SE}%MKUKATPVW %CVW_SPS %VBOASG %P 2:F327 = AUS, 3: BOASG
         $FLAG[327] = FALSE
      ;ENDFOLD
      ;FOLD F329 = AUS ;%{SE}%MKUKATPVW %CVW_SPS %VBOASG %P 2:F329 = AUS, 3: BOASG
         $FLAG[329] = FALSE
      ;ENDFOLD
      ;FOLD -- EZ1/SP1/KE1 SZ3 Zaehler -- ;%{SE}%MKUKATPVW %CVW_COM %VCOMMENT %P 2:-- EZ1/SP1/KE1 SZ3 Zaehler --, 3: VW_COMMENT
      ;ENDFOLD
      ;FOLD F106 = AUS ;%{SE}%MKUKATPVW %CVW_SPS %VBOASG %P 2:F106 = AUS, 3: BOASG
         $FLAG[106] = FALSE
      ;ENDFOLD
      ;FOLD F107 = AUS ;%{SE}%MKUKATPVW %CVW_SPS %VBOASG %P 2:F107 = AUS, 3: BOASG
         $FLAG[107] = FALSE
      ;ENDFOLD
      ;FOLD F108 = AUS ;%{SE}%MKUKATPVW %CVW_SPS %VBOASG %P 2:F108 = AUS, 3: BOASG
         $FLAG[108] = FALSE
      ;ENDFOLD
      ;FOLD F109 = AUS ;%{SE}%MKUKATPVW %CVW_SPS %VBOASG %P 2:F109 = AUS, 3: BOASG
         $FLAG[109] = FALSE
      ;ENDFOLD
      ;FOLD F110 = AUS ;%{SE}%MKUKATPVW %CVW_SPS %VBOASG %P 2:F110 = AUS, 3: BOASG
         $FLAG[110] = FALSE
      ;ENDFOLD
      ;FOLD F111 = AUS ;%{SE}%MKUKATPVW %CVW_SPS %VBOASG %P 2:F111 = AUS, 3: BOASG
         $FLAG[111] = FALSE
      ;ENDFOLD
      ;FOLD -- Hilfsflags Funktionstest KF Motor -- ;%{SE}%MKUKATPVW %CVW_COM %VCOMMENT %P 2:-- Hilfsflags Funktionstest KF Motor --, 3: VW_COMMENT
      ;ENDFOLD
      ;FOLD F312 = AUS ;%{SE}%MKUKATPVW %CVW_SPS %VBOASG %P 2:F312 = AUS, 3: BOASG
         $FLAG[312] = FALSE
      ;ENDFOLD
      ;FOLD F313 = AUS ;%{SE}%MKUKATPVW %CVW_SPS %VBOASG %P 2:F313 = AUS, 3: BOASG
         $FLAG[313] = FALSE
      ;ENDFOLD
      ;FOLD -- Rob. EZ1/SP1 SZ3 beim Fraesen -- ;%{SE}%MKUKATPVW %CVW_COM %VCOMMENT %P 2:-- Rob. EZ1/SP1 SZ3 beim Fraesen --, 3: VW_COMMENT
      ;ENDFOLD
      ;FOLD A116 = EIN ;%{SE}%MKUKATPVW %CVW_SPS %VBOASG %P 2:A116 = EIN, 3: BOASG
         $OUT[116] = TRUE
      ;ENDFOLD
      ;FOLD A130 = EIN ;%{SE}%MKUKATPVW %CVW_SPS %VBOASG %P 2:A130 = EIN, 3: BOASG
         $OUT[130] = TRUE
      ;ENDFOLD
      ;FOLD -- Quitt. Fraesen SK1 AUS -- ;%{SE}%MKUKATPVW %CVW_COM %VCOMMENT %P 2:-- Quitt. Fraesen SK1 AUS --, 3: VW_COMMENT
      ;ENDFOLD
      ;FOLD A786 = F830 & A786 ;%{SE}%MKUKATPVW %CVW_SPS %VBOASG %P 2:A786 = F830 & A786, 3: BOASG
         $OUT[786] = $FLAG[830] AND $OUT[786]
      ;ENDFOLD
      ;FOLD A722 = !F830 & A722 ;%{SE}%MKUKATPVW %CVW_SPS %VBOASG %P 2:A722 = !F830 & A722, 3: BOASG
         $OUT[722] = NOT $FLAG[830] AND $OUT[722]
      ;ENDFOLD
      ;FOLD -- Ueberwachungszeit KF1/KW1 -- ;%{SE}%MKUKATPVW %CVW_COM %VCOMMENT %P 2:-- Ueberwachungszeit KF1/KW1 --, 3: VW_COMMENT
      ;ENDFOLD
      ;FOLD t7 ( EIN ) = -30[1/10Sek] ;%{SE}%MKUKATPVW %CVW_SPS %VTASG %P 2:t7 ( EIN ) = -30[1/10Sek], 3: TASG
         VW(#SET_TIME,TRUE,7,0,-30)
      ;ENDFOLD
      ;FOLD Schritt 28 = A4039  ;%{SE}%MKUKATPVW %CVW_SPS %VST_CON %P 2:Schritt 28 = A4039 , 3: ST_CON
         IF $OUT[4039] THEN
            PREVSTEP = $APP_INT[5]
            $APP_INT[5] = 28
         ENDIF
      ;ENDFOLD
   ;ENDFOLD
   ;FOLD SCHRITT 28 -- ROB EZ1/SP1/KE1 SZ3 -- ;%{P}%MKUKATPVW,%CSTEP,%VST_NR,%P 1:SCHRITT, 2:28, 3: ROB EZ1/SP1/KE1 SZ3
      ;FOLD ;%{H}
         Case 28
      ;ENDFOLD
      ;FOLD -- KF1/KW1 einschalten -- ;%{SE}%MKUKATPVW %CVW_COM %VCOMMENT %P 2:-- KF1/KW1 einschalten --, 3: VW_COMMENT
      ;ENDFOLD
      ;FOLD i1 (EIN) = 0 ;%{SE}%MKUKATPVW %CVW_SPS %VARIASG %P 2:i1 (EIN) = 0, 3: ARIASG
         VW(#COUNTER,TRUE,1,0)
      ;ENDFOLD
      ;FOLD A834 = !F289 ;%{SE}%MKUKATPVW %CVW_SPS %VBOASG %P 2:A834 = !F289, 3: BOASG
         $OUT[834] = NOT $FLAG[289]
      ;ENDFOLD
      ;FOLD A858 = F289 ;%{SE}%MKUKATPVW %CVW_SPS %VBOASG %P 2:A858 = F289, 3: BOASG
         $OUT[858] = $FLAG[289]
      ;ENDFOLD
      ;FOLD A1018 = F803 ;%{SE}%MKUKATPVW %CVW_SPS %VBOASG %P 2:A1018 = F803, 3: BOASG
         $OUT[1018] = $FLAG[803]
      ;ENDFOLD
      ;FOLD Schritt 29 = A4039  ;%{SE}%MKUKATPVW %CVW_SPS %VST_CON %P 2:Schritt 29 = A4039 , 3: ST_CON
         IF $OUT[4039] THEN
            PREVSTEP = $APP_INT[5]
            $APP_INT[5] = 29
         ENDIF
      ;ENDFOLD
   ;ENDFOLD
   ;FOLD SCHRITT 29 -- ROB EZ1/SP1/KE1 SZ3 -- ;%{P}%MKUKATPVW,%CSTEP,%VST_NR,%P 1:SCHRITT, 2:29, 3: ROB EZ1/SP1/KE1 SZ3
      ;FOLD ;%{H}
         Case 29
      ;ENDFOLD
      ;FOLD -- Funktionstest KF Motor -- ;%{SE}%MKUKATPVW %CVW_COM %VCOMMENT %P 2:-- Funktionstest KF Motor --, 3: VW_COMMENT
      ;ENDFOLD
      ;FOLD F312 = EIN ;%{SE}%MKUKATPVW %CVW_SPS %VBOASG %P 2:F312 = EIN, 3: BOASG
         $FLAG[312] = TRUE
      ;ENDFOLD
      ;FOLD F313 = i1 > 2 ;%{SE}%MKUKATPVW %CVW_SPS %VBOCMP %P 2:F313 = i1 > 2, 3: BOCMP
         $FLAG[313] = $COUNT_I[1] > 2
      ;ENDFOLD
      ;FOLD Schritt 30 = (F313 + T7) & A4039  ;%{SE}%MKUKATPVW %CVW_SPS %VST_CON %P 2:Schritt 30 = (F313 + T7) & A4039 , 3: ST_CON
